KUKA KRL program: MyProgram_181().src

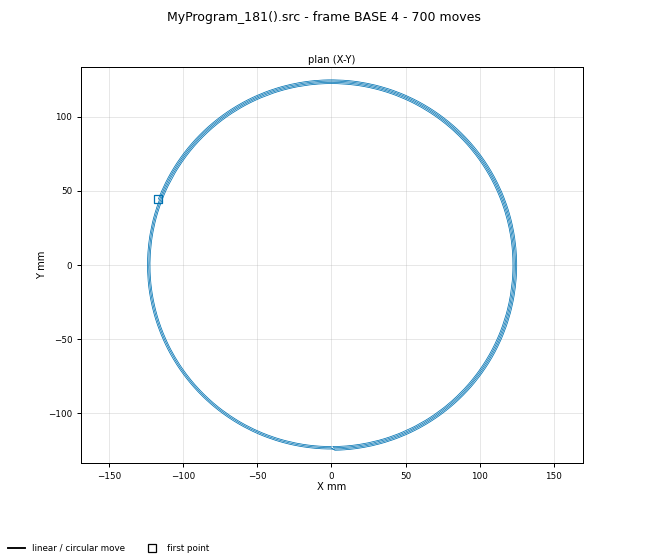
[picture p0: tool path of MyProgram_181().src in frame BASE 4, 700 of 700 moves have a stored position in this frame; points joined in program order, loops and branches not executed]
&ACCESS RVP
&REL 1
&PARAM TEMPLATE = C:\KRC\Roboter\Template\vorgabe
&PARAM EDITMASK = *
DEF MyProgram_181()
; ---- Setting reference (Base) ----
$BASE = BASE_DATA[4]

; --------------------------
; ---- Setting tool (TCP) ----
$TOOL = TOOL_DATA[3]
; --------------------------

$VEL.CP = VEL_APROX_PRINT
Startdeposition()
$VEL.CP = VEL_PRINT
LIN {X -116.6895,Y 44.4583,Z 133,A 155.0312,B 24.9522,C -1.5964,E1 24.8506,E2 291.2943} C_DIS
LIN {X -115.697,Y 46.9762,Z 133,A 153.7111,B 24.9522,C -1.5969,E1 24.852,E2 292.6207} C_DIS
LIN {X -114.3662,Y 50.133,Z 133,A 152.1883,B 24.9518,C -1.6039,E1 24.8537,E2 294.1352} C_DIS
LIN {X -113.0397,Y 53.0574,Z 133,A 150.686,B 24.9516,C -1.6071,E1 24.8554,E2 295.638} C_DIS
LIN {X -111.9021,Y 55.4109,Z 133,A 149.4421,B 24.9516,C -1.6088,E1 24.857,E2 296.8845} C_DIS
LIN {X -110.1873,Y 58.7517,Z 133,A 147.6606,B 24.9513,C -1.6113,E1 24.8593,E2 298.6696} C_DIS
LIN {X -108.2507,Y 62.2485,Z 133,A 145.7452,B 24.9513,C -1.6131,E1 24.8619,E2 300.5907} C_DIS
LIN {X -105.81,Y 66.3134,Z 133,A 143.6874,B 24.9505,C -1.6247,E1 24.8649,E2 302.6316} C_DIS
LIN {X -103.9306,Y 69.2193,Z 133,A 142.0204,B 24.9505,C -1.6257,E1 24.8675,E2 304.3045} C_DIS
LIN {X -101.3647,Y 72.9272,Z 133,A 139.999,B 24.95,C -1.6336,E1 24.8707,E2 306.317} C_DIS
LIN {X -99.2695,Y 75.7526,Z 133,A 138.3169,B 24.95,C -1.635,E1 24.8735,E2 308.0039} C_DIS
LIN {X -96.6511,Y 79.0667,Z 133,A 136.3828,B 24.9496,C -1.6403,E1 24.8769,E2 309.9343} C_DIS
LIN {X -94.1983,Y 81.973,Z 133,A 134.6073,B 24.9494,C -1.6435,E1 24.8801,E2 311.7102} C_DIS
LIN {X -91.6588,Y 84.8038,Z 133,A 132.8618,B 24.9491,C -1.648,E1 24.8834,E2 313.4528} C_DIS
LIN {X -88.8677,Y 87.7247,Z 133,A 130.926,B 24.9491,C -1.6489,E1 24.8872,E2 315.3948} C_DIS
LIN {X -86.0086,Y 90.5292,Z 133,A 129.1473,B 24.9486,C -1.656,E1 24.8907,E2 317.164} C_DIS
LIN {X -83.0096,Y 93.2873,Z 133,A 127.2009,B 24.9486,C -1.6569,E1 24.8948,E2 319.1159} C_DIS
LIN {X -79.9792,Y 95.8975,Z 133,A 125.4366,B 24.9481,C -1.6643,E1 24.8985,E2 320.8696} C_DIS
LIN {X -76.816,Y 98.4502,Z 133,A 123.4845,B 24.9481,C -1.6644,E1 24.9028,E2 322.8286} C_DIS
LIN {X -73.6345,Y 100.8511,Z 133,A 121.7327,B 24.9476,C -1.6718,E1 24.9067,E2 324.5692} C_DIS
LIN {X -70.3577,Y 103.1645,Z 133,A 119.7925,B 24.9476,C -1.671,E1 24.9112,E2 326.5178} C_DIS
LIN {X -66.9879,Y 105.3831,Z 133,A 118.0307,B 24.9472,C -1.6786,E1 24.9153,E2 328.267} C_DIS
LIN {X -63.5914,Y 107.4674,Z 133,A 116.1028,B 24.9472,C -1.6775,E1 24.9199,E2 330.2036} C_DIS
LIN {X -59.4752,Y 109.7995,Z 133,A 113.9327,B 24.947,C -1.6814,E1 24.9252,E2 332.3708} C_DIS
LIN {X -56.3954,Y 111.4096,Z 133,A 112.4464,B 24.9465,C -1.689,E1 24.9289,E2 333.8429} C_DIS
LIN {X -53.3186,Y 112.9163,Z 133,A 110.9027,B 24.9463,C -1.6928,E1 24.9327,E2 335.3817} C_DIS
LIN {X -50.4991,Y 114.2045,Z 133,A 109.4916,B 24.9461,C -1.6955,E1 24.9363,E2 336.7898} C_DIS
LIN {X -47.5925,Y 115.4458,Z 133,A 108.05,B 24.946,C -1.698,E1 24.94,E2 338.2288} C_DIS
LIN {X -44.9062,Y 116.5167,Z 133,A 106.6465,B 24.946,C -1.6963,E1 24.9437,E2 339.6392} C_DIS
LIN {X -41.647,Y 117.7232,Z 133,A 105.0866,B 24.9458,C -1.6999,E1 24.9478,E2 341.1937} C_DIS
LIN {X -38.7891,Y 118.6945,Z 133,A 103.7405,B 24.9456,C -1.7034,E1 24.9513,E2 342.534} C_DIS
LIN {X -36.2059,Y 119.5067,Z 133,A 102.4321,B 24.9457,C -1.7018,E1 24.9548,E2 343.8484} C_DIS
LIN {X -32.9677,Y 120.4422,Z 133,A 100.9122,B 24.9455,C -1.7047,E1 24.9589,E2 345.3639} C_DIS
LIN {X -29.9898,Y 121.2171,Z 133,A 99.5473,B 24.9453,C -1.7083,E1 24.9626,E2 346.7223} C_DIS
LIN {X -27.3572,Y 121.8375,Z 133,A 98.2908,B 24.9453,C -1.7087,E1 24.966,E2 347.9793} C_DIS
LIN {X -24.1727,Y 122.5102,Z 133,A 96.8162,B 24.9451,C -1.7109,E1 24.97,E2 349.4506} C_DIS
LIN {X -21.6943,Y 122.9714,Z 133,A 95.5852,B 24.9453,C -1.7083,E1 24.9734,E2 350.6889} C_DIS
LIN {X -18.3848,Y 123.5119,Z 133,A 94.0677,B 24.9452,C -1.7103,E1 24.9776,E2 352.203} C_DIS
LIN {X -14.9172,Y 123.9758,Z 133,A 92.4267,B 24.9452,C -1.7097,E1 24.9822,E2 353.8466} C_DIS
LIN {X -11.5107,Y 124.3398,Z 133,A 90.8991,B 24.945,C -1.7126,E1 24.9864,E2 355.3683} C_DIS
LIN {X -8.4462,Y 124.5859,Z 133,A 89.5189,B 24.945,C -1.7146,E1 24.9902,E2 356.7442} C_DIS
LIN {X -5.7492,Y 124.7393,Z 133,A 88.2519,B 24.945,C -1.7138,E1 24.9938,E2 358.0135} C_DIS
LIN {X -2.325,Y 124.8487,Z 133,A 86.6375,B 24.945,C -1.7122,E1 24.9983,E2 359.6318} C_DIS
LIN {X 1.3218,Y 124.8654,Z 133,A 84.8045,B 24.9455,C -1.705,E1 25.0034,E2 361.4819} C_DIS
LIN {X 5.505,Y 124.7509,Z 133,A 83.1157,B 24.9448,C -1.7161,E1 25.0081,E2 363.144} C_DIS
LIN {X 8.0461,Y 124.6112,Z 133,A 81.7359,B 24.9455,C -1.7061,E1 25.012,E2 364.5469} C_DIS
LIN {X 11.9921,Y 124.2936,Z 133,A 80.0376,B 24.9451,C -1.7115,E1 25.0167,E2 366.2314} C_DIS
LIN {X 14.8682,Y 123.9817,Z 133,A 78.6941,B 24.9451,C -1.7105,E1 25.0204,E2 367.5763} C_DIS
LIN {X 18.2642,Y 123.5297,Z 133,A 77.174,B 24.9451,C -1.7125,E1 25.0246,E2 369.0903} C_DIS
LIN {X 21.2737,Y 123.0464,Z 133,A 75.8309,B 24.9449,C -1.7147,E1 25.0283,E2 370.4269} C_DIS
LIN {X 23.9077,Y 122.5611,Z 133,A 74.5912,B 24.9449,C -1.7137,E1 25.0317,E2 371.6675} C_DIS
LIN {X 27.0788,Y 121.9008,Z 133,A 73.1177,B 24.9449,C -1.7135,E1 25.0357,E2 373.1395} C_DIS
LIN {X 29.5009,Y 121.3353,Z 133,A 71.8951,B 24.9453,C -1.709,E1 25.039,E2 374.3711} C_DIS
LIN {X 32.8189,Y 120.4825,Z 133,A 70.3477,B 24.9453,C -1.7091,E1 25.0432,E2 375.9158} C_DIS
LIN {X 35.8156,Y 119.6254,Z 133,A 68.9731,B 24.9452,C -1.7108,E1 25.0469,E2 377.2842} C_DIS
LIN {X 38.3543,Y 118.8346,Z 133,A 67.6655,B 24.9455,C -1.7056,E1 25.0504,E2 378.6015} C_DIS
LIN {X 41.6005,Y 117.7396,Z 133,A 66.1321,B 24.9455,C -1.706,E1 25.0544,E2 380.1309} C_DIS
LIN {X 44.4583,Y 116.6895,Z 133,A 64.7708,B 24.9455,C -1.7064,E1 25.058,E2 381.4883} C_DIS
LIN {X 46.9533,Y 115.7063,Z 133,A 63.4699,B 24.9457,C -1.7018,E1 25.0614,E2 382.7974} C_DIS
LIN {X 50.1104,Y 114.376,Z 133,A 61.9635,B 24.9457,C -1.7032,E1 25.0652,E2 384.2968} C_DIS
LIN {X 53.0574,Y 113.0397,Z 133,A 60.4644,B 24.9457,C -1.7007,E1 25.069,E2 385.798} C_DIS
LIN {X 55.4907,Y 111.8627,Z 133,A 59.2079,B 24.9459,C -1.6984,E1 25.0722,E2 387.0566} C_DIS
LIN {X 58.7517,Y 110.1873,Z 133,A 57.4722,B 24.9463,C -1.6935,E1 25.0765,E2 388.7991} C_DIS
LIN {X 62.2484,Y 108.2507,Z 133,A 55.5685,B 24.9466,C -1.6874,E1 25.0811,E2 390.7114} C_DIS
LIN {X 66.3133,Y 105.81,Z 133,A 53.5313,B 24.9464,C -1.6909,E1 25.086,E2 392.7341} C_DIS
LIN {X 69.2398,Y 103.9169,Z 133,A 51.8763,B 24.9468,C -1.6855,E1 25.0898,E2 394.3963} C_DIS
LIN {X 72.9272,Y 101.3646,Z 133,A 49.8782,B 24.9468,C -1.6849,E1 25.0944,E2 396.389} C_DIS
LIN {X 75.7723,Y 99.2545,Z 133,A 48.2058,B 24.9471,C -1.6796,E1 25.0981,E2 398.0676} C_DIS
LIN {X 79.3312,Y 96.4353,Z 133,A 46.1821,B 24.9471,C -1.6786,E1 25.1025,E2 400.0862} C_DIS
LIN {X 81.9916,Y 94.1821,Z 133,A 44.5325,B 24.9476,C -1.673,E1 25.106,E2 401.7426} C_DIS
LIN {X 84.8038,Y 91.6588,Z 133,A 42.8054,B 24.9478,C -1.6697,E1 25.1096,E2 403.4705} C_DIS
LIN {X 87.7247,Y 88.8677,Z 133,A 40.8925,B 24.9482,C -1.6628,E1 25.1135,E2 405.3917} C_DIS
LIN {X 90.5292,Y 86.0086,Z 133,A 39.1388,B 24.9482,C -1.6629,E1 25.1168,E2 407.1376} C_DIS
LIN {X 93.2873,Y 83.0096,Z 133,A 37.2042,B 24.9487,C -1.6554,E1 25.1205,E2 409.0814} C_DIS
LIN {X 95.8975,Y 79.9792,Z 133,A 35.4643,B 24.9487,C -1.6558,E1 25.1236,E2 410.8124} C_DIS
LIN {X 98.4502,Y 76.816,Z 133,A 33.5535,B 24.949,C -1.6489,E1 25.1269,E2 412.7304} C_DIS
LIN {X 100.8511,Y 73.6345,Z 133,A 31.7966,B 24.9491,C -1.648,E1 25.1299,E2 414.4812} C_DIS
LIN {X 103.1645,Y 70.3577,Z 133,A 29.8671,B 24.9497,C -1.6387,E1 25.1329,E2 416.423} C_DIS
LIN {X 105.3831,Y 66.9879,Z 133,A 28.1306,B 24.9497,C -1.6396,E1 25.1356,E2 418.1487} C_DIS
LIN {X 107.4674,Y 63.5914,Z 133,A 26.2144,B 24.9502,C -1.6303,E1 25.1383,E2 420.0772} C_DIS
LIN {X 109.8114,Y 59.4535,Z 133,A 24.0555,B 24.9505,C -1.6254,E1 25.1413,E2 422.2363} C_DIS
LIN {X 112.1236,Y 54.9624,Z 133,A 21.8943,B 24.9505,C -1.6268,E1 25.144,E2 424.3827} C_DIS
LIN {X 113.6675,Y 51.6979,Z 133,A 20.282,B 24.9505,C -1.6243,E1 25.1459,E2 425.9923} C_DIS
LIN {X 114.7933,Y 49.1453,Z 133,A 18.9532,B 24.9509,C -1.618,E1 25.1474,E2 427.3284} C_DIS
LIN {X 116.0423,Y 46.1217,Z 133,A 17.4924,B 24.9511,C -1.6156,E1 25.1489,E2 428.7869} C_DIS
LIN {X 117.2068,Y 43.0763,Z 133,A 16.052,B 24.9511,C -1.614,E1 25.1503,E2 430.2232} C_DIS
LIN {X 118.0998,Y 40.5602,Z 133,A 14.7553,B 24.9516,C -1.6066,E1 25.1515,E2 431.5298} C_DIS
LIN {X 119.0422,Y 37.7053,Z 133,A 13.4155,B 24.9518,C -1.6044,E1 25.1526,E2 432.8673} C_DIS
LIN {X 120.0332,Y 34.4239,Z 133,A 11.8937,B 24.9519,C -1.6022,E1 25.1538,E2 434.3858} C_DIS
LIN {X 121.0581,Y 30.6172,Z 133,A 10.0158,B 24.9525,C -1.593,E1 25.1552,E2 436.2744} C_DIS
LIN {X 121.8429,Y 27.3332,Z 133,A 8.5584,B 24.9525,C -1.5928,E1 25.1561,E2 437.7237} C_DIS
LIN {X 122.5102,Y 24.1727,Z 133,A 7.1037,B 24.9527,C -1.5895,E1 25.1569,E2 439.1778} C_DIS
LIN {X 122.9405,Y 21.8675,Z 133,A 5.9294,B 24.9532,C -1.5811,E1 25.1575,E2 440.3651} C_DIS
LIN {X 123.5119,Y 18.3848,Z 133,A 4.398,B 24.9532,C -1.5803,E1 25.1582,E2 441.8892} C_DIS
LIN {X 124.0763,Y 14.0747,Z 133,A 2.4493,B 24.9534,C -1.5763,E1 25.1589,E2 443.836} C_DIS
LIN {X 124.3421,Y 11.4861,Z 133,A 1.2276,B 24.9538,C -1.571,E1 25.1592,E2 445.063} C_DIS
LIN {X 124.5859,Y 8.4462,Z 133,A -0.1347,B 24.9539,C -1.5683,E1 25.1595,E2 446.4235} C_DIS
LIN {X 124.7483,Y 5.5668,Z 133,A -1.6675,B 24.9548,C -1.5532,E1 25.1597,E2 447.9827} C_DIS
LIN {X 124.8637,Y 1.4441,Z 133,A -3.3231,B 24.9545,C -1.5592,E1 25.1597,E2 449.6145} C_DIS
LIN {X 124.8646,Y -1.3828,Z 133,A -4.8305,B 24.9553,C -1.5441,E1 25.1597,E2 451.1484} C_DIS
LIN {X 124.7508,Y -5.505,Z 133,A -6.489,B 24.955,C -1.5499,E1 25.1596,E2 452.7834} C_DIS
LIN {X 124.5347,Y -9.1442,Z 133,A -8.2497,B 24.9556,C -1.5399,E1 25.1593,E2 454.5571} C_DIS
LIN {X 124.2394,Y -12.5574,Z 133,A -9.7621,B 24.9556,C -1.5378,E1 25.1589,E2 456.0656} C_DIS
LIN {X 123.9788,Y -14.8927,Z 133,A -10.8875,B 24.956,C -1.5318,E1 25.1585,E2 457.1984} C_DIS
LIN {X 123.5851,Y -17.8742,Z 133,A -12.2192,B 24.9562,C -1.5298,E1 25.158,E2 458.5271} C_DIS
LIN {X 123.1574,Y -20.6093,Z 133,A -13.5143,B 24.9565,C -1.5243,E1 25.1574,E2 459.8274} C_DIS
LIN {X 122.5658,Y -23.8834,Z 133,A -14.9527,B 24.9565,C -1.5239,E1 25.1567,E2 461.2584} C_DIS
LIN {X 121.9008,Y -27.0788,Z 133,A -16.4252,B 24.9567,C -1.5203,E1 25.1558,E2 462.731} C_DIS
LIN {X 121.3295,Y -29.5249,Z 133,A -17.6476,B 24.9571,C -1.513,E1 25.155,E2 463.9634} C_DIS
LIN {X 120.5319,Y -32.6336,Z 133,A -19.0811,B 24.9573,C -1.5102,E1 25.154,E2 465.3953} C_DIS
LIN {X 119.6254,Y -35.8156,Z 133,A -20.5468,B 24.9573,C -1.508,E1 25.1529,E2 466.8578} C_DIS
LIN {X 118.8421,Y -38.3307,Z 133,A -21.838,B 24.9579,C -1.4999,E1 25.1518,E2 468.1606} C_DIS
LIN {X 117.7477,Y -41.5771,Z 133,A -23.3597,B 24.9579,C -1.4975,E1 25.1504,E2 469.6795} C_DIS
LIN {X 116.6895,Y -44.4583,Z 133,A -24.7286,B 24.9581,C -1.4951,E1 25.1491,E2 471.0464} C_DIS
LIN {X 115.697,Y -46.9762,Z 133,A -25.9971,B 24.9584,C -1.4898,E1 25.1477,E2 472.3203} C_DIS
LIN {X 114.3662,Y -50.133,Z 133,A -27.5341,B 24.9586,C -1.4867,E1 25.146,E2 473.8562} C_DIS
LIN {X 113.0397,Y -53.0574,Z 133,A -29.0168,B 24.9589,C -1.4817,E1 25.1443,E2 475.3427} C_DIS
LIN {X 111.924,Y -55.3666,Z 133,A -30.2101,B 24.9591,C -1.4773,E1 25.1428,E2 476.5399} C_DIS
LIN {X 110.1873,Y -58.7517,Z 133,A -32.0034,B 24.9595,C -1.4696,E1 25.1405,E2 478.3421} C_DIS
LIN {X 108.2507,Y -62.2485,Z 133,A -33.8947,B 24.96,C -1.4612,E1 25.1379,E2 480.2432} C_DIS
LIN {X 105.81,Y -66.3134,Z 133,A -35.9274,B 24.96,C -1.4621,E1 25.1349,E2 482.2634} C_DIS
LIN {X 103.9306,Y -69.2193,Z 133,A -37.5741,B 24.9604,C -1.4546,E1 25.1324,E2 483.9196} C_DIS
LIN {X 101.3647,Y -72.9272,Z 133,A -39.5716,B 24.9604,C -1.4524,E1 25.1292,E2 485.9125} C_DIS
LIN {X 99.2695,Y -75.7526,Z 133,A -41.234,B 24.9609,C -1.4455,E1 25.1264,E2 487.5834} C_DIS
LIN {X 96.4353,Y -79.3313,Z 133,A -43.2607,B 24.9609,C -1.4433,E1 25.1229,E2 489.6059} C_DIS
LIN {X 94.1983,Y -81.973,Z 133,A -44.9018,B 24.9613,C -1.4364,E1 25.1199,E2 491.2556} C_DIS
LIN {X 91.6588,Y -84.8038,Z 133,A -46.6283,B 24.9615,C -1.4328,E1 25.1166,E2 492.9829} C_DIS
LIN {X 88.8677,Y -87.7247,Z 133,A -48.5435,B 24.962,C -1.4251,E1 25.1129,E2 494.9082} C_DIS
LIN {X 86.0086,Y -90.5292,Z 133,A -50.304,B 24.962,C -1.4245,E1 25.1093,E2 496.6629} C_DIS
LIN {X 83.0096,Y -93.2873,Z 133,A -52.2308,B 24.9624,C -1.4171,E1 25.1053,E2 498.5992} C_DIS
LIN {X 79.9792,Y -95.8975,Z 133,A -53.9782,B 24.9624,C -1.4174,E1 25.1016,E2 500.3393} C_DIS
LIN {X 76.816,Y -98.4502,Z 133,A -55.9119,B 24.9628,C -1.4097,E1 25.0974,E2 502.2837} C_DIS
LIN {X 73.6345,Y -100.8511,Z 133,A -57.6481,B 24.9628,C -1.4105,E1 25.0935,E2 504.012} C_DIS
LIN {X 70.3577,Y -103.1645,Z 133,A -59.5713,B 24.9632,C -1.4025,E1 25.0891,E2 505.9473} C_DIS
LIN {X 66.9879,Y -105.3831,Z 133,A -61.3186,B 24.9631,C -1.4041,E1 25.085,E2 507.6852} C_DIS
LIN {X 63.5914,Y -107.4674,Z 133,A -63.231,B 24.9635,C -1.3964,E1 25.0804,E2 509.6099} C_DIS
LIN {X 59.4752,Y -109.7995,Z 133,A -65.3847,B 24.9636,C -1.3934,E1 25.0751,E2 511.7645} C_DIS
LIN {X 56.3954,Y -111.4096,Z 133,A -66.8606,B 24.9635,C -1.3966,E1 25.0715,E2 513.2286} C_DIS
LIN {X 53.3186,Y -112.9163,Z 133,A -68.3983,B 24.9635,C -1.3957,E1 25.0676,E2 514.7644} C_DIS
LIN {X 50.2713,Y -114.3064,Z 133,A -69.9153,B 24.9635,C -1.3943,E1 25.0637,E2 516.281} C_DIS
LIN {X 47.4675,Y -115.498,Z 133,A -71.2814,B 24.9636,C -1.3938,E1 25.0602,E2 517.6449} C_DIS
LIN {X 44.9062,Y -116.5167,Z 133,A -72.6234,B 24.9639,C -1.3882,E1 25.0567,E2 518.9972} C_DIS
LIN {X 41.647,Y -117.7232,Z 133,A -74.1722,B 24.9639,C -1.3883,E1 25.0527,E2 520.5426} C_DIS
LIN {X 38.7891,Y -118.6945,Z 133,A -75.5018,B 24.9639,C -1.3894,E1 25.0492,E2 521.8673} C_DIS
LIN {X 36.2059,Y -119.5067,Z 133,A -76.8155,B 24.9641,C -1.3844,E1 25.0456,E2 523.1904} C_DIS
LIN {X 32.9677,Y -120.4422,Z 133,A -78.3284,B 24.9641,C -1.3843,E1 25.0416,E2 524.701} C_DIS
LIN {X 29.9898,Y -121.2171,Z 133,A -79.6875,B 24.9641,C -1.3854,E1 25.0379,E2 526.0553} C_DIS
LIN {X 27.3572,Y -121.8375,Z 133,A -80.9389,B 24.9641,C -1.3837,E1 25.0345,E2 527.309} C_DIS
LIN {X 24.1727,Y -122.5102,Z 133,A -82.4081,B 24.9641,C -1.3836,E1 25.0305,E2 528.7767} C_DIS
LIN {X 21.6943,Y -122.9714,Z 133,A -83.6348,B 24.9644,C -1.3792,E1 25.0271,E2 530.0124} C_DIS
LIN {X 18.6063,Y -123.4775,Z 133,A -85.0343,B 24.9644,C -1.3799,E1 25.0232,E2 531.4089} C_DIS
LIN {X 16.0341,Y -123.8366,Z 133,A -86.203,B 24.9644,C -1.3803,E1 25.02,E2 532.5757} C_DIS
LIN {X 12.7087,Y -124.2243,Z 133,A -87.7444,B 24.9644,C -1.3791,E1 25.0157,E2 534.119} C_DIS
LIN {X 8.6784,Y -124.5689,Z 133,A -89.5972,B 24.9644,C -1.3783,E1 25.0105,E2 535.9725} C_DIS
LIN {X 5.7492,Y -124.7393,Z 133,A -90.9508,B 24.9644,C -1.3774,E1 25.0068,E2 537.3279} C_DIS
LIN {X 2.325,Y -124.8487,Z 133,A -92.5631,B 24.9646,C -1.375,E1 25.0023,E2 538.9456} C_DIS
LIN {X 2.325,Y -124.8487,Z 133,A -92.5631,B 24.9646,C -1.375,E1 25.0023,E2 538.9456} C_DIS
Enddeposition()
LIN {X 0.8859,Y -124.0293,Z 133,A -93.2093,B 24.9638,C -1.3903,E1 25.0006,E2 539.5556} C_DIS
Startdeposition()
$VEL.CP = VEL_PRINT
LIN {X 3.5558,Y -123.9822,Z 133,A -91.4139,B 24.9623,C -1.4178,E1 25.0058,E2 537.6952} C_DIS
LIN {X 6.3715,Y -123.8705,Z 133,A -90.0135,B 24.9621,C -1.4231,E1 25.0097,E2 536.2827} C_DIS
LIN {X 9.98,Y -123.6317,Z 133,A -88.2827,B 24.9619,C -1.4268,E1 25.0145,E2 534.5439} C_DIS
LIN {X 13.8144,Y -123.2627,Z 133,A -86.4414,B 24.9616,C -1.4309,E1 25.0197,E2 532.6943} C_DIS
LIN {X 17.6544,Y -122.7711,Z 133,A -84.7834,B 24.9619,C -1.4257,E1 25.0242,E2 531.0499} C_DIS
LIN {X 21.7768,Y -122.1067,Z 133,A -82.9831,B 24.9622,C -1.4208,E1 25.0291,E2 529.2629} C_DIS
LIN {X 24.7936,Y -121.5298,Z 133,A -81.504,B 24.962,C -1.425,E1 25.0332,E2 527.7757} C_DIS
LIN {X 27.7732,Y -120.8845,Z 133,A -80.0201,B 24.9617,C -1.4301,E1 25.0373,E2 526.2818} C_DIS
LIN {X 31.1769,Y -120.0529,Z 133,A -78.1591,B 24.961,C -1.4438,E1 25.0424,E2 524.3912} C_DIS
LIN {X 34.9694,Y -119.0013,Z 133,A -76.6182,B 24.9616,C -1.4321,E1 25.0464,E2 522.8806} C_DIS
LIN {X 38.0799,Y -118.0438,Z 133,A -74.9694,B 24.9611,C -1.4411,E1 25.0509,E2 521.2135} C_DIS
LIN {X 41.8289,Y -116.7678,Z 133,A -73.2082,B 24.9611,C -1.4401,E1 25.0555,E2 519.4582} C_DIS
LIN {X 45.1339,Y -115.5304,Z 133,A -71.6275,B 24.9611,C -1.4399,E1 25.0596,E2 517.8814} C_DIS
LIN {X 48.4667,Y -114.1737,Z 133,A -69.8642,B 24.9608,C -1.4474,E1 25.0642,E2 516.1045} C_DIS
LIN {X 52.5572,Y -112.3489,Z 133,A -67.8625,B 24.9608,C -1.4473,E1 25.0693,E2 514.1081} C_DIS
LIN {X 57.0107,Y -110.1577,Z 133,A -65.6711,B 24.9608,C -1.446,E1 25.0747,E2 511.9256} C_DIS
LIN {X 61.6993,Y -107.6005,Z 133,A -62.7982,B 24.9595,C -1.471,E1 25.0818,E2 509.0022} C_DIS
LIN {X 64.8534,Y -105.729,Z 133,A -61.5813,B 24.9606,C -1.4501,E1 25.0846,E2 507.8386} C_DIS
LIN {X 67.8771,Y -103.8154,Z 133,A -59.3711,B 24.9589,C -1.4816,E1 25.09,E2 505.5612} C_DIS
LIN {X 71.2509,Y -101.528,Z 133,A -58.093,B 24.9604,C -1.4547,E1 25.0927,E2 504.3509} C_DIS
LIN {X 74.1934,Y -99.3988,Z 133,A -56.216,B 24.9596,C -1.4684,E1 25.097,E2 502.4483} C_DIS
LIN {X 77.4252,Y -96.9017,Z 133,A -54.1352,B 24.9588,C -1.4825,E1 25.1016,E2 500.342} C_DIS
LIN {X 79.9254,Y -94.8499,Z 133,A -52.8711,B 24.9593,C -1.4742,E1 25.1043,E2 499.1023} C_DIS
LIN {X 83.1574,Y -92.0304,Z 133,A -50.8978,B 24.9591,C -1.4784,E1 25.1084,E2 497.1269} C_DIS
LIN {X 86.6144,Y -88.7849,Z 133,A -48.4884,B 24.9581,C -1.4949,E1 25.1133,E2 494.6885} C_DIS
LIN {X 88.9161,Y -86.4791,Z 133,A -46.7364,B 24.9572,C -1.5115,E1 25.1168,E2 492.905} C_DIS
LIN {X 92.0187,Y -83.1704,Z 133,A -45.3655,B 24.959,C -1.4797,E1 25.1192,E2 491.6153} C_DIS
LIN {X 94.2078,Y -80.6831,Z 133,A -43.5512,B 24.9579,C -1.4982,E1 25.1226,E2 489.7654} C_DIS
LIN {X 99.1932,Y -74.4686,Z 133,A -40.0644,B 24.9579,C -1.4982,E1 25.1286,E2 486.2949} C_DIS
LIN {X 101.1843,Y -71.7386,Z 133,A -38.3986,B 24.9574,C -1.508,E1 25.1313,E2 484.6141} C_DIS
LIN {X 103.7575,Y -67.9649,Z 133,A -36.2868,B 24.9571,C -1.5141,E1 25.1346,E2 482.4984} C_DIS
LIN {X 106.0577,Y -64.3145,Z 133,A -34.3457,B 24.9569,C -1.5172,E1 25.1374,E2 480.5598} C_DIS
LIN {X 108.866,Y -59.4378,Z 133,A -31.7507,B 24.9564,C -1.5247,E1 25.141,E2 477.9607} C_DIS
LIN {X 110.4663,Y -56.4043,Z 133,A -30.2235,B 24.9564,C -1.5266,E1 25.143,E2 476.4372} C_DIS
LIN {X 112.1094,Y -53.0661,Z 133,A -28.5971,B 24.9564,C -1.527,E1 25.1449,E2 474.8184} C_DIS
LIN {X 113.5497,Y -49.9129,Z 133,A -26.7086,B 24.9552,C -1.5468,E1 25.1471,E2 472.8936} C_DIS
LIN {X 115.0838,Y -46.2601,Z 133,A -25.1254,B 24.9556,C -1.5398,E1 25.1488,E2 471.3356} C_DIS
LIN {X 116.5902,Y -42.3211,Z 133,A -22.5573,B 24.9533,C -1.5781,E1 25.1513,E2 468.6914} C_DIS
LIN {X 118.1658,Y -37.6984,Z 133,A -21.1923,B 24.9556,C -1.5391,E1 25.1524,E2 467.4263} C_DIS
LIN {X 118.947,Y -35.1547,Z 133,A -19.7275,B 24.9547,C -1.5552,E1 25.1536,E2 465.9319} C_DIS
LIN {X 119.9648,Y -31.5112,Z 133,A -17.7372,B 24.9536,C -1.5734,E1 25.1551,E2 463.9101} C_DIS
LIN {X 120.9703,Y -27.3964,Z 133,A -15.9606,B 24.9538,C -1.5704,E1 25.1562,E2 462.1509} C_DIS
LIN {X 121.9265,Y -22.7744,Z 133,A -13.9465,B 24.9538,C -1.5689,E1 25.1573,E2 460.1521} C_DIS
LIN {X 122.3948,Y -20.0956,Z 133,A -12.7048,B 24.9537,C -1.5723,E1 25.1578,E2 458.9097} C_DIS
LIN {X 122.9518,Y -16.3453,Z 133,A -10.6973,B 24.9526,C -1.5913,E1 25.1586,E2 456.8692} C_DIS
LIN {X 123.3707,Y -12.8176,Z 133,A -9.1701,B 24.9526,C -1.5907,E1 25.1591,E2 455.3523} C_DIS
LIN {X 123.6944,Y -9.1605,Z 133,A -7.5598,B 24.9526,C -1.5919,E1 25.1594,E2 453.7488} C_DIS
LIN {X 123.9124,Y -5.5254,Z 133,A -5.79,B 24.9519,C -1.6019,E1 25.1597,E2 451.9659} C_DIS
LIN {X 124.0303,Y -1.1139,Z 133,A -3.8363,B 24.9518,C -1.6042,E1 25.1597,E2 450.0185} C_DIS
LIN {X 124.0095,Y 2.4534,Z 133,A -2.3173,B 24.9518,C -1.603,E1 25.1597,E2 448.5114} C_DIS
LIN {X 123.8912,Y 5.9529,Z 133,A -0.6589,B 24.9514,C -1.6104,E1 25.1595,E2 446.8453} C_DIS
LIN {X 123.6626,Y 9.5941,Z 133,A 1.0564,B 24.951,C -1.6174,E1 25.1592,E2 445.1237} C_DIS
LIN {X 123.3513,Y 12.9962,Z 133,A 2.4302,B 24.9513,C -1.612,E1 25.1588,E2 443.7707} C_DIS
LIN {X 123.0151,Y 15.8622,Z 133,A 3.8699,B 24.9507,C -1.6218,E1 25.1583,E2 442.3164} C_DIS
LIN {X 122.5217,Y 19.3088,Z 133,A 5.486,B 24.9504,C -1.6274,E1 25.1577,E2 440.6967} C_DIS
LIN {X 121.7898,Y 23.4864,Z 133,A 7.9703,B 24.9483,C -1.6608,E1 25.1564,E2 438.1482} C_DIS
LIN {X 120.9086,Y 27.6672,Z 133,A 9.3663,B 24.9498,C -1.6372,E1 25.1556,E2 436.8161} C_DIS
LIN {X 120.1497,Y 30.7951,Z 133,A 10.8555,B 24.9495,C -1.642,E1 25.1545,E2 435.3241} C_DIS
LIN {X 118.7254,Y 35.899,Z 133,A 13.3527,B 24.9489,C -1.652,E1 25.1526,E2 432.8175} C_DIS
LIN {X 117.6528,Y 39.2679,Z 133,A 14.9177,B 24.9488,C -1.6536,E1 25.1513,E2 431.2578} C_DIS
LIN {X 116.6813,Y 42.0688,Z 133,A 16.3181,B 24.9484,C -1.6593,E1 25.1499,E2 429.8518} C_DIS
LIN {X 115.5152,Y 45.1731,Z 133,A 17.8908,B 24.948,C -1.6659,E1 25.1484,E2 428.2722} C_DIS
LIN {X 114.0858,Y 48.6732,Z 133,A 19.6391,B 24.9477,C -1.6711,E1 25.1465,E2 426.5211} C_DIS
LIN {X 111.4188,Y 54.4996,Z 133,A 22.6482,B 24.947,C -1.6822,E1 25.1429,E2 423.5022} C_DIS
LIN {X 109.803,Y 57.6851,Z 133,A 24.1283,B 24.9472,C -1.6782,E1 25.141,E2 422.0395} C_DIS
LIN {X 107.8139,Y 61.3259,Z 133,A 26.1659,B 24.9465,C -1.6896,E1 25.1382,E2 419.9855} C_DIS
LIN {X 105.4931,Y 65.2374,Z 133,A 28.175,B 24.9465,C -1.6906,E1 25.1353,E2 417.9843} C_DIS
LIN {X 103.3371,Y 68.6012,Z 133,A 30.0123,B 24.9462,C -1.695,E1 25.1325,E2 416.1457} C_DIS
LIN {X 101.1257,Y 71.8217,Z 133,A 31.5892,B 24.9466,C -1.6881,E1 25.13,E2 414.5928} C_DIS
LIN {X 99.16,Y 74.5126,Z 133,A 33.4363,B 24.9454,C -1.7076,E1 25.1269,E2 412.7087} C_DIS
LIN {X 93.8986,Y 81.0415,Z 133,A 36.8985,B 24.9461,C -1.6961,E1 25.1209,E2 409.2896} C_DIS
LIN {X 91.4285,Y 83.8176,Z 133,A 38.9118,B 24.9449,C -1.715,E1 25.117,E2 407.2408} C_DIS
LIN {X 88.6849,Y 86.7162,Z 133,A 40.7508,B 24.9446,C -1.7188,E1 25.1135,E2 405.4005} C_DIS
LIN {X 82.3107,Y 92.788,Z 133,A 44.6184,B 24.9447,C -1.7173,E1 25.1057,E2 401.5525} C_DIS
LIN {X 79.577,Y 95.1425,Z 133,A 46.4597,B 24.944,C -1.7293,E1 25.1017,E2 399.69} C_DIS
LIN {X 76.428,Y 97.6907,Z 133,A 48.2789,B 24.9439,C -1.7302,E1 25.0977,E2 397.8754} C_DIS
LIN {X 73.4502,Y 99.9481,Z 133,A 50.0816,B 24.9434,C -1.7371,E1 25.0937,E2 396.0628} C_DIS
LIN {X 69.884,Y 102.4746,Z 133,A 52.0902,B 24.9433,C -1.74,E1 25.0891,E2 394.0543} C_DIS
LIN {X 66.4489,Y 104.734,Z 133,A 53.9827,B 24.9431,C -1.7428,E1 25.0846,E2 392.1615} C_DIS
LIN {X 62.6592,Y 107.044,Z 133,A 55.885,B 24.9434,C -1.7386,E1 25.0801,E2 390.275} C_DIS
LIN {X 59.275,Y 108.9551,Z 133,A 57.8558,B 24.9426,C -1.7498,E1 25.0752,E2 388.2835} C_DIS
LIN {X 55.3777,Y 110.9852,Z 133,A 59.9211,B 24.9423,C -1.7542,E1 25.0701,E2 386.2134} C_DIS
LIN {X 51.3378,Y 112.9119,Z 133,A 61.7646,B 24.9429,C -1.7456,E1 25.0655,E2 384.3947} C_DIS
LIN {X 48.3344,Y 114.229,Z 133,A 63.5089,B 24.942,C -1.7586,E1 25.0609,E2 382.6241} C_DIS
LIN {X 43.9336,Y 115.9923,Z 133,A 65.5764,B 24.9423,C -1.7548,E1 25.0556,E2 380.5701} C_DIS
LIN {X 40.1406,Y 117.3595,Z 133,A 67.3385,B 24.9425,C -1.7516,E1 25.051,E2 378.8192} C_DIS
LIN {X 34.3616,Y 119.1794,Z 133,A 70.0646,B 24.9425,C -1.7502,E1 25.0437,E2 376.1013} C_DIS
LIN {X 31.5406,Y 119.957,Z 133,A 71.7954,B 24.9413,C -1.7694,E1 25.0389,E2 374.3276} C_DIS
LIN {X 26.7398,Y 121.1179,Z 133,A 73.8442,B 24.942,C -1.7594,E1 25.0334,E2 372.3054} C_DIS
LIN {X 22.9306,Y 121.8965,Z 133,A 75.5899,B 24.942,C -1.7577,E1 25.0287,E2 370.5657} C_DIS
LIN {X 18.4276,Y 122.6584,Z 133,A 77.6255,B 24.9423,C -1.7549,E1 25.0231,E2 368.5388} C_DIS
LIN {X 15.0746,Y 123.1143,Z 133,A 79.2629,B 24.942,C -1.7588,E1 25.0185,E2 366.8934} C_DIS
LIN {X 11.716,Y 123.4794,Z 133,A 80.8193,B 24.942,C -1.7588,E1 25.0142,E2 365.3381} C_DIS
LIN {X 8.3403,Y 123.7544,Z 133,A 82.526,B 24.9416,C -1.7657,E1 25.0094,E2 363.6159} C_DIS
LIN {X 5.0114,Y 123.9324,Z 133,A 83.9197,B 24.942,C -1.7586,E1 25.0056,E2 362.2394} C_DIS
LIN {X 1.0086,Y 124.0303,Z 133,A 85.7913,B 24.942,C -1.7594,E1 25.0003,E2 360.3661} C_DIS
LIN {X -2.6617,Y 124.006,Z 133,A 87.5064,B 24.942,C -1.7599,E1 24.9955,E2 358.6498} C_DIS
LIN {X -6.6373,Y 123.8573,Z 133,A 89.4432,B 24.9417,C -1.764,E1 24.9901,E2 356.7029} C_DIS
LIN {X -10.7031,Y 123.571,Z 133,A 91.253,B 24.942,C -1.7597,E1 24.9851,E2 354.9025} C_DIS
LIN {X -14.7477,Y 123.1533,Z 133,A 93.0653,B 24.9422,C -1.7555,E1 24.9801,E2 353.0989} C_DIS
LIN {X -19.7935,Y 122.4452,Z 133,A 95.3399,B 24.9426,C -1.7502,E1 24.9738,E2 350.8351} C_DIS
LIN {X -28.1635,Y 120.7956,Z 133,A 99.3624,B 24.9426,C -1.7506,E1 24.9628,E2 346.807} C_DIS
LIN {X -32.338,Y 119.7446,Z 133,A 101.5073,B 24.9422,C -1.7559,E1 24.957,E2 344.6464} C_DIS
LIN {X -36.19,Y 118.6364,Z 133,A 103.3087,B 24.9425,C -1.7515,E1 24.9522,E2 342.8524} C_DIS
LIN {X -40.4709,Y 117.2451,Z 133,A 105.9696,B 24.9409,C -1.776,E1 24.945,E2 340.1281} C_DIS
LIN {X -45.0709,Y 115.5549,Z 133,A 107.5069,B 24.9433,C -1.7392,E1 24.9412,E2 338.6751} C_DIS
LIN {X -47.4506,Y 114.5982,Z 133,A 108.8036,B 24.9431,C -1.7426,E1 24.9378,E2 337.3673} C_DIS
LIN {X -50.8002,Y 113.1529,Z 133,A 110.7175,B 24.9426,C -1.7507,E1 24.9329,E2 335.4297} C_DIS
LIN {X -55.1327,Y 111.1062,Z 133,A 112.6255,B 24.9437,C -1.733,E1 24.9282,E2 333.5587} C_DIS
LIN {X -58.5811,Y 109.3294,Z 133,A 114.5844,B 24.9434,C -1.7376,E1 24.9233,E2 331.5834} C_DIS
LIN {X -62.257,Y 107.2783,Z 133,A 116.4586,B 24.9438,C -1.7309,E1 24.9188,E2 329.7197} C_DIS
LIN {X -65.6502,Y 105.2367,Z 133,A 118.4096,B 24.9438,C -1.733,E1 24.9141,E2 327.7576} C_DIS
LIN {X -69.5314,Y 102.7131,Z 133,A 120.4881,B 24.9442,C -1.7261,E1 24.9093,E2 325.6888} C_DIS
LIN {X -72.9755,Y 100.2956,Z 133,A 122.4562,B 24.9444,C -1.7232,E1 24.9048,E2 323.7208} C_DIS
LIN {X -76.5034,Y 97.6315,Z 133,A 124.5347,B 24.9445,C -1.7204,E1 24.9002,E2 321.6412} C_DIS
LIN {X -79.6512,Y 95.0802,Z 133,A 126.3504,B 24.945,C -1.7137,E1 24.8963,E2 319.8347} C_DIS
LIN {X -82.9389,Y 92.2273,Z 133,A 128.4243,B 24.945,C -1.7119,E1 24.892,E2 317.7569} C_DIS
LIN {X -86.074,Y 89.3079,Z 133,A 130.3916,B 24.9454,C -1.7066,E1 24.888,E2 315.7939} C_DIS
LIN {X -89.092,Y 86.2974,Z 133,A 132.3606,B 24.9457,C -1.7018,E1 24.8841,E2 313.8282} C_DIS
LIN {X -92.0675,Y 83.1168,Z 133,A 134.4273,B 24.9459,C -1.6991,E1 24.8802,E2 311.7587} C_DIS
LIN {X -94.7666,Y 80.0249,Z 133,A 136.3261,B 24.9462,C -1.6943,E1 24.8768,E2 309.8627} C_DIS
LIN {X -97.4905,Y 76.6829,Z 133,A 138.3002,B 24.9466,C -1.6881,E1 24.8733,E2 307.894} C_DIS
LIN {X -99.9533,Y 73.4431,Z 133,A 140.1542,B 24.947,C -1.6818,E1 24.8703,E2 306.0461} C_DIS
LIN {X -102.5748,Y 69.7362,Z 133,A 142.226,B 24.9474,C -1.6748,E1 24.867,E2 303.9809} C_DIS
LIN {X -104.5452,Y 66.7449,Z 133,A 143.885,B 24.9477,C -1.6703,E1 24.8644,E2 302.3242} C_DIS
LIN {X -106.7152,Y 63.2189,Z 133,A 145.8353,B 24.948,C -1.6664,E1 24.8616,E2 300.3732} C_DIS
LIN {X -108.4898,Y 60.1209,Z 133,A 147.467,B 24.9483,C -1.6608,E1 24.8594,E2 298.7463} C_DIS
LIN {X -110.1607,Y 57.005,Z 133,A 149.4146,B 24.9477,C -1.6699,E1 24.8568,E2 296.7667} C_DIS
LIN {X -112.0866,Y 53.1137,Z 133,A 151.0986,B 24.949,C -1.6495,E1 24.8548,E2 295.1222} C_DIS
LIN {X -113.3254,Y 50.4146,Z 133,A 152.5167,B 24.9491,C -1.6473,E1 24.8532,E2 293.7014} C_DIS
LIN {X -115.0123,Y 46.4369,Z 133,A 154.5962,B 24.9493,C -1.6449,E1 24.851,E2 291.6162} C_DIS
LIN {X -116.4149,Y 42.8047,Z 133,A 156.4474,B 24.9495,C -1.6415,E1 24.8492,E2 289.7625} C_DIS
LIN {X -117.6385,Y 39.3108,Z 133,A 158.11,B 24.95,C -1.634,E1 24.8477,E2 288.1083} C_DIS
LIN {X -119.0141,Y 34.9257,Z 133,A 160.1791,B 24.9505,C -1.6249,E1 24.846,E2 286.0492} C_DIS
LIN {X -119.9113,Y 31.7122,Z 133,A 161.706,B 24.9509,C -1.6193,E1 24.8449,E2 284.5267} C_DIS
LIN {X -120.7064,Y 28.5408,Z 133,A 163.4001,B 24.9507,C -1.6225,E1 24.8437,E2 282.815} C_DIS
LIN {X -122.1749,Y 21.3941,Z 133,A 166.5462,B 24.9519,C -1.6016,E1 24.8421,E2 279.7002} C_DIS
LIN {X -122.6148,Y 18.709,Z 133,A 168.178,B 24.9512,C -1.6141,E1 24.8413,E2 278.0288} C_DIS
LIN {X -123.1938,Y 14.4073,Z 133,A 169.8826,B 24.9524,C -1.5942,E1 24.8408,E2 276.3614} C_DIS
LIN {X -123.5038,Y 11.4615,Z 133,A 171.3058,B 24.9525,C -1.5921,E1 24.8404,E2 274.9347} C_DIS
LIN {X -123.7427,Y 8.5024,Z 133,A 172.8011,B 24.9525,C -1.5931,E1 24.8401,E2 273.4279} C_DIS
LIN {X -124.0018,Y 2.8572,Z 133,A 175.4499,B 24.9529,C -1.5863,E1 24.8398,E2 270.7796} C_DIS
LIN {X -123.9758,Y -3.7863,Z 133,A 177.9877,B 24.9548,C -1.5527,E1 24.8398,E2 268.3066} C_DIS
LIN {X -123.5574,Y -10.8648,Z 133,A -178.3715,B 24.9545,C -1.5581,E1 24.8405,E2 264.631} C_DIS
LIN {X -123.1186,Y -15.0385,Z 133,A -176.045,B 24.9539,C -1.5691,E1 24.8412,E2 262.2642} C_DIS
LIN {X -122.6875,Y -18.2394,Z 133,A -174.2558,B 24.9534,C -1.5776,E1 24.842,E2 260.4441} C_DIS
LIN {X -121.9566,Y -22.617,Z 133,A -172.6072,B 24.9548,C -1.5531,E1 24.8428,E2 258.8442} C_DIS
LIN {X -121.1902,Y -26.4046,Z 133,A -171.0469,B 24.9557,C -1.5374,E1 24.8437,E2 257.312} C_DIS
LIN {X -120.5423,Y -29.2196,Z 133,A -169.5819,B 24.9557,C -1.5391,E1 24.8446,E2 255.8345} C_DIS
LIN {X -119.4404,Y -33.4404,Z 133,A -167.5917,B 24.956,C -1.5317,E1 24.8461,E2 253.8503} C_DIS
LIN {X -118.4229,Y -36.8885,Z 133,A -165.9534,B 24.9564,C -1.5256,E1 24.8474,E2 252.2172} C_DIS
LIN {X -117.2471,Y -40.4654,Z 133,A -164.0338,B 24.9562,C -1.5284,E1 24.8491,E2 250.2799} C_DIS
LIN {X -115.9273,Y -44.1074,Z 133,A -162.4347,B 24.957,C -1.5145,E1 24.8506,E2 248.705} C_DIS
LIN {X -114.938,Y -46.6209,Z 133,A -161.0572,B 24.957,C -1.5167,E1 24.8521,E2 247.3146} C_DIS
LIN {X -112.9855,Y -51.1742,Z 133,A -158.8591,B 24.9575,C -1.5059,E1 24.8545,E2 245.13} C_DIS
LIN {X -111.6547,Y -54.0166,Z 133,A -157.4106,B 24.9578,C -1.5017,E1 24.8563,E2 243.6837} C_DIS
LIN {X -110.1929,Y -56.9422,Z 133,A -155.4283,B 24.9568,C -1.5187,E1 24.8589,E2 241.6502} C_DIS
LIN {X -108.5221,Y -60.0626,Z 133,A -154.1511,B 24.958,C -1.498,E1 24.8605,E2 240.4157} C_DIS
LIN {X -106.4779,Y -63.6172,Z 133,A -152.163,B 24.958,C -1.4971,E1 24.8634,E2 238.4194} C_DIS
LIN {X -104.0433,Y -67.5253,Z 133,A -150.1273,B 24.9586,C -1.4873,E1 24.8664,E2 236.3966} C_DIS
LIN {X -101.995,Y -70.582,Z 133,A -148.3617,B 24.9586,C -1.4859,E1 24.8692,E2 234.6256} C_DIS
LIN {X -99.5933,Y -73.9313,Z 133,A -146.424,B 24.9588,C -1.4827,E1 24.8724,E2 232.6862} C_DIS
LIN {X -97.1423,Y -77.1235,Z 133,A -144.5828,B 24.9591,C -1.4773,E1 24.8755,E2 230.849} C_DIS
LIN {X -95.1088,Y -79.6171,Z 133,A -143.0885,B 24.9593,C -1.4742,E1 24.8782,E2 229.3554} C_DIS
LIN {X -92.4643,Y -82.6742,Z 133,A -141.2223,B 24.9595,C -1.4698,E1 24.8816,E2 227.4912} C_DIS
LIN {X -89.8184,Y -85.5411,Z 133,A -139.3872,B 24.9597,C -1.4673,E1 24.8851,E2 225.6541} C_DIS
LIN {X -86.6754,Y -88.725,Z 133,A -137.3281,B 24.9599,C -1.4625,E1 24.8892,E2 223.5977} C_DIS
LIN {X -83.9889,Y -91.2712,Z 133,A -135.8392,B 24.9607,C -1.4488,E1 24.8922,E2 222.1353} C_DIS
LIN {X -81.8219,Y -93.2193,Z 133,A -134.2902,B 24.9603,C -1.4554,E1 24.8955,E2 220.5644} C_DIS
LIN {X -79.0019,Y -95.6211,Z 133,A -132.5823,B 24.9605,C -1.452,E1 24.8991,E2 218.8581} C_DIS
LIN {X -76.0446,Y -97.9892,Z 133,A -130.6123,B 24.9601,C -1.4589,E1 24.9035,E2 216.8643} C_DIS
LIN {X -73.0539,Y -100.2386,Z 133,A -129.078,B 24.9608,C -1.4469,E1 24.9069,E2 215.3532} C_DIS
LIN {X -69.8763,Y -102.4798,Z 133,A -127.1585,B 24.9606,C -1.4496,E1 24.9113,E2 213.4208} C_DIS
LIN {X -65.9,Y -105.0816,Z 133,A -125.1093,B 24.9612,C -1.4393,E1 24.9161,E2 211.3895} C_DIS
LIN {X -62.9754,Y -106.8585,Z 133,A -123.4309,B 24.9611,C -1.4415,E1 24.9202,E2 209.7006} C_DIS
LIN {X -59.1297,Y -109.0346,Z 133,A -121.3706,B 24.9611,C -1.4396,E1 24.9252,E2 207.6391} C_DIS
LIN {X -55.6937,Y -110.8274,Z 133,A -119.743,B 24.9617,C -1.4297,E1 24.9292,E2 206.0306} C_DIS
LIN {X -53.2727,Y -112.0105,Z 133,A -118.387,B 24.9615,C -1.4334,E1 24.9326,E2 204.6623} C_DIS
LIN {X -49.1048,Y -113.8991,Z 133,A -116.3983,B 24.962,C -1.4251,E1 24.9377,E2 202.6884} C_DIS
LIN {X -46.4796,Y -114.9951,Z 133,A -114.9503,B 24.9617,C -1.4301,E1 24.9414,E2 201.2254} C_DIS
LIN {X -43.3333,Y -116.217,Z 133,A -113.4345,B 24.9619,C -1.4266,E1 24.9454,E2 199.7147} C_DIS
LIN {X -37.2584,Y -118.3065,Z 133,A -110.3895,B 24.9619,C -1.4277,E1 24.9535,E2 196.6613} C_DIS
LIN {X -33.0845,Y -119.5403,Z 133,A -108.362,B 24.9619,C -1.4272,E1 24.9589,E2 194.6318} C_DIS
LIN {X -28.5875,Y -120.6952,Z 133,A -106.3338,B 24.9622,C -1.4204,E1 24.9644,E2 192.6169} C_DIS
LIN {X -25.4958,Y -121.3863,Z 133,A -104.8711,B 24.9622,C -1.4197,E1 24.9684,E2 191.1541} C_DIS
LIN {X -21.6486,Y -122.1295,Z 133,A -103.1397,B 24.9625,C -1.4152,E1 24.9731,E2 189.4314} C_DIS
LIN {X -18.7892,Y -122.6023,Z 133,A -101.6907,B 24.9622,C -1.4201,E1 24.9771,E2 187.9694} C_DIS
LIN {X -15.1656,Y -123.1035,Z 133,A -99.8823,B 24.9619,C -1.4255,E1 24.9822,E2 186.1469} C_DIS
LIN {X -11.3696,Y -123.5126,Z 133,A -98.0548,B 24.9618,C -1.4284,E1 24.9873,E2 184.3115} C_DIS
LIN {X -6.7538,Y -123.8515,Z 133,A -95.9549,B 24.9618,C -1.4266,E1 24.9931,E2 182.2152} C_DIS
LIN {X -2.7431,Y -124.0046,Z 133,A -94.1605,B 24.962,C -1.424,E1 24.9981,E2 180.4268} C_DIS
LIN {X 0.8859,Y -124.0293,Z 133,A -93.2073,B 24.9638,C -1.3894,E1 25.0006,E2 179.5556} C_DIS
Enddeposition()
LIN {X 0.8859,Y -124.0293,Z 133,A -93.2073,B 24.9638,C -1.3894,E1 25.0006,E2 179.5556} C_DIS
Startdeposition()
$VEL.CP = VEL_PRINT
LIN {X -0.0675,Y -123.1989,Z 133,A -93.8487,B 24.9636,C -1.3946,E1 24.9988,E2 180.1847} C_DIS
LIN {X -4.2619,Y -123.1237,Z 133,A -95.792,B 24.9636,C -1.3946,E1 24.9934,E2 182.128} C_DIS
LIN {X -8.2359,Y -122.9224,Z 133,A -97.7799,B 24.9639,C -1.3881,E1 24.9878,E2 184.132} C_DIS
LIN {X -13.016,Y -122.5074,Z 133,A -99.8282,B 24.9634,C -1.397,E1 24.9821,E2 186.1606} C_DIS
LIN {X -16.9419,Y -122.0271,Z 133,A -101.547,B 24.9631,C -1.403,E1 24.9774,E2 187.8663} C_DIS
LIN {X -20.4358,Y -121.4895,Z 133,A -103.6369,B 24.9642,C -1.3826,E1 24.9715,E2 190.0064} C_DIS
LIN {X -23.9849,Y -120.8404,Z 133,A -105.0446,B 24.9635,C -1.3959,E1 24.9677,E2 191.3843} C_DIS
LIN {X -27.768,Y -120.0274,Z 133,A -106.8977,B 24.9635,C -1.3942,E1 24.9627,E2 193.2436} C_DIS
LIN {X -32.936,Y -118.7127,Z 133,A -109.2782,B 24.9633,C -1.4004,E1 24.9563,E2 195.613} C_DIS
LIN {X -36.7255,Y -117.5977,Z 133,A -111.2666,B 24.9636,C -1.3947,E1 24.9509,E2 197.6184} C_DIS
LIN {X -41.3333,Y -116.0571,Z 133,A -113.406,B 24.9632,C -1.4022,E1 24.9453,E2 199.7441} C_DIS
LIN {X -44.5175,Y -114.8721,Z 133,A -114.8926,B 24.9629,C -1.408,E1 24.9415,E2 201.2199} C_DIS
LIN {X -47.9326,Y -113.4899,Z 133,A -117.1212,B 24.964,C -1.3862,E1 24.9356,E2 203.5055} C_DIS
LIN {X -51.5883,Y -111.8745,Z 133,A -118.4018,B 24.9625,C -1.4148,E1 24.9325,E2 204.7212} C_DIS
LIN {X -53.9087,Y -110.7773,Z 133,A -119.9704,B 24.9633,C -1.399,E1 24.9284,E2 206.3314} C_DIS
LIN {X -58.7842,Y -108.2697,Z 133,A -122.3855,B 24.9628,C -1.4086,E1 24.9225,E2 208.7305} C_DIS
LIN {X -62.8547,Y -105.958,Z 133,A -124.55,B 24.9626,C -1.4123,E1 24.9173,E2 210.8926} C_DIS
LIN {X -67.9729,Y -102.7495,Z 133,A -127.3512,B 24.9624,C -1.4171,E1 24.9107,E2 213.6914} C_DIS
LIN {X -70.3817,Y -101.1143,Z 133,A -129.2871,B 24.9636,C -1.3931,E1 24.9062,E2 215.6908} C_DIS
LIN {X -74.3909,Y -98.2027,Z 133,A -131.029,B 24.9621,C -1.4225,E1 24.9024,E2 217.3692} C_DIS
LIN {X -77.046,Y -96.1337,Z 133,A -132.555,B 24.9618,C -1.4272,E1 24.899,E2 218.8897} C_DIS
LIN {X -80.2936,Y -93.4385,Z 133,A -134.5549,B 24.9618,C -1.4293,E1 24.8948,E2 220.8922} C_DIS
LIN {X -83.3607,Y -90.7119,Z 133,A -136.694,B 24.9621,C -1.4229,E1 24.8903,E2 223.0553} C_DIS
LIN {X -85.7027,Y -88.5029,Z 133,A -137.9344,B 24.9613,C -1.4375,E1 24.8879,E2 224.2659} C_DIS
LIN {X -88.4807,Y -85.7257,Z 133,A -139.7507,B 24.961,C -1.442,E1 24.8843,E2 226.0793} C_DIS
LIN {X -91.3836,Y -82.6249,Z 133,A -141.6385,B 24.9606,C -1.4503,E1 24.8808,E2 227.9556} C_DIS
LIN {X -93.6332,Y -80.0675,Z 133,A -143.4428,B 24.9609,C -1.4442,E1 24.8774,E2 229.7828} C_DIS
LIN {X -96.6554,Y -76.3913,Z 133,A -145.6135,B 24.9605,C -1.4514,E1 24.8736,E2 231.9464} C_DIS
LIN {X -98.982,Y -73.3508,Z 133,A -147.4018,B 24.9603,C -1.4555,E1 24.8706,E2 233.7335} C_DIS
LIN {X -101.4047,Y -69.9638,Z 133,A -149.3866,B 24.9602,C -1.4583,E1 24.8674,E2 235.7213} C_DIS
LIN {X -103.1148,Y -67.4195,Z 133,A -151.2295,B 24.961,C -1.4437,E1 24.8646,E2 237.6084} C_DIS
LIN {X -105.3382,Y -63.8871,Z 133,A -152.4058,B 24.9588,C -1.4826,E1 24.863,E2 238.698} C_DIS
LIN {X -109.281,Y -56.8802,Z 133,A -156.5747,B 24.9593,C -1.4738,E1 24.8573,E2 242.9096} C_DIS
LIN {X -111.0088,Y -53.4275,Z 133,A -158.2069,B 24.9586,C -1.4861,E1 24.8553,E2 244.5215} C_DIS
LIN {X -112.0597,Y -51.1873,Z 133,A -160.0047,B 24.96,C -1.4612,E1 24.8531,E2 246.3884} C_DIS
LIN {X -113.9565,Y -46.8154,Z 133,A -162.4507,B 24.9602,C -1.4578,E1 24.8505,E2 248.8562} C_DIS
LIN {X -115.9958,Y -41.503,Z 133,A -164.7093,B 24.9588,C -1.4825,E1 24.8484,E2 251.0687} C_DIS
LIN {X -117.2268,Y -37.8871,Z 133,A -166.0842,B 24.9575,C -1.5054,E1 24.8472,E2 252.3969} C_DIS
LIN {X -118.2899,Y -34.4212,Z 133,A -167.7946,B 24.9573,C -1.5095,E1 24.8459,E2 254.1074} C_DIS
LIN {X -119.3648,Y -30.4857,Z 133,A -169.6705,B 24.9569,C -1.5163,E1 24.8445,E2 255.9779} C_DIS
LIN {X -120.1619,Y -27.1773,Z 133,A -171.3815,B 24.9569,C -1.5157,E1 24.8434,E2 257.7004} C_DIS
LIN {X -121.1422,Y -22.418,Z 133,A -173.6675,B 24.9566,C -1.5217,E1 24.8422,E2 259.9857} C_DIS
LIN {X -121.8709,Y -18.0409,Z 133,A -175.5445,B 24.9558,C -1.5364,E1 24.8414,E2 261.8387} C_DIS
LIN {X -122.5901,Y -12.2222,Z 133,A -179.2038,B 24.9576,C -1.505,E1 24.8403,E2 265.5948} C_DIS
LIN {X -123.0259,Y -6.5057,Z 133,A 179.1058,B 24.9547,C -1.5557,E1 24.84,E2 267.1745} C_DIS
LIN {X -123.1923,Y -1.2278,Z 133,A 176.3454,B 24.955,C -1.5505,E1 24.8398,E2 269.964} C_DIS
LIN {X -122.9836,Y 7.2542,Z 133,A 172.458,B 24.9541,C -1.566,E1 24.8402,E2 273.8378} C_DIS
LIN {X -122.7675,Y 10.2704,Z 133,A 170.8354,B 24.9543,C -1.5613,E1 24.8405,E2 275.4815} C_DIS
LIN {X -121.9895,Y 17.2064,Z 133,A 167.8694,B 24.953,C -1.584,E1 24.8415,E2 278.411} C_DIS
LIN {X -121.4566,Y 20.6326,Z 133,A 166.3751,B 24.9524,C -1.5944,E1 24.8422,E2 279.8894} C_DIS
LIN {X -120.9106,Y 23.6231,Z 133,A 164.5109,B 24.9533,C -1.5795,E1 24.8431,E2 281.8002} C_DIS
LIN {X -119.8594,Y 28.4831,Z 133,A 162.3826,B 24.9523,C -1.5949,E1 24.8444,E2 283.9042} C_DIS
LIN {X -118.9681,Y 32.0019,Z 133,A 160.7071,B 24.952,C -1.6009,E1 24.8456,E2 285.5752} C_DIS
LIN {X -118.0746,Y 35.1562,Z 133,A 158.947,B 24.9523,C -1.5956,E1 24.847,E2 287.3581} C_DIS
LIN {X -116.5435,Y 39.9398,Z 133,A 157.0598,B 24.9507,C -1.6225,E1 24.8486,E2 289.1921} C_DIS
LIN {X -115.5384,Y 42.759,Z 133,A 155.4281,B 24.951,C -1.6164,E1 24.8502,E2 290.8474} C_DIS
LIN {X -114.3724,Y 45.7869,Z 133,A 153.8224,B 24.951,C -1.617,E1 24.8519,E2 292.4608} C_DIS
LIN {X -112.8949,Y 49.3187,Z 133,A 152.0301,B 24.9507,C -1.6219,E1 24.8538,E2 294.2512} C_DIS
LIN {X -111.2716,Y 52.8782,Z 133,A 150.4858,B 24.9496,C -1.6395,E1 24.8556,E2 295.7621} C_DIS
LIN {X -108.5552,Y 58.2542,Z 133,A 147.4843,B 24.9496,C -1.6391,E1 24.8595,E2 298.7806} C_DIS
LIN {X -106.7558,Y 61.4899,Z 133,A 145.6576,B 24.9496,C -1.6396,E1 24.862,E2 300.6156} C_DIS
LIN {X -104.3555,Y 65.4824,Z 133,A 143.5003,B 24.9492,C -1.6463,E1 24.8651,E2 302.7681} C_DIS
LIN {X -100.901,Y 70.6877,Z 133,A 140.5901,B 24.9487,C -1.6543,E1 24.8697,E2 305.6737} C_DIS
LIN {X -98.5323,Y 73.9552,Z 133,A 138.6192,B 24.9487,C -1.6553,E1 24.8729,E2 307.6516} C_DIS
LIN {X -95.6199,Y 77.6831,Z 133,A 136.4728,B 24.9481,C -1.6636,E1 24.8766,E2 309.7884} C_DIS
LIN {X -93.0468,Y 80.747,Z 133,A 134.6014,B 24.9479,C -1.668,E1 24.88,E2 311.6578} C_DIS
LIN {X -90.0818,Y 84.0422,Z 133,A 132.5127,B 24.9476,C -1.6721,E1 24.884,E2 313.7461} C_DIS
LIN {X -87.2368,Y 86.9911,Z 133,A 130.6556,B 24.9472,C -1.6789,E1 24.8876,E2 315.5948} C_DIS
LIN {X -84.1602,Y 89.9722,Z 133,A 128.5543,B 24.9472,C -1.6789,E1 24.8919,E2 317.7048} C_DIS
LIN {X -80.8101,Y 92.9918,Z 133,A 126.5511,B 24.9466,C -1.688,E1 24.896,E2 319.6945} C_DIS
LIN {X -77.7744,Y 95.5454,Z 133,A 124.6522,B 24.9465,C -1.6897,E1 24.9001,E2 321.5964} C_DIS
LIN {X -74.3663,Y 98.2213,Z 133,A 122.6434,B 24.9462,C -1.6943,E1 24.9045,E2 323.6016} C_DIS
LIN {X -71.1711,Y 100.5604,Z 133,A 120.7765,B 24.946,C -1.697,E1 24.9088,E2 325.4685} C_DIS
LIN {X -67.3324,Y 103.1714,Z 133,A 118.8488,B 24.9451,C -1.7116,E1 24.9132,E2 327.368} C_DIS
LIN {X -64.1213,Y 105.196,Z 133,A 116.8816,B 24.9455,C -1.706,E1 24.9179,E2 329.3548} C_DIS
LIN {X -60.6374,Y 107.2428,Z 133,A 114.9382,B 24.9455,C -1.7065,E1 24.9226,E2 331.3027} C_DIS
LIN {X -56.6936,Y 109.3792,Z 133,A 112.9057,B 24.945,C -1.7124,E1 24.9276,E2 333.3267} C_DIS
LIN {X -53.9438,Y 110.7599,Z 133,A 111.1445,B 24.9458,C -1.7,E1 24.9321,E2 335.1221} C_DIS
LIN {X -50.8496,Y 112.2139,Z 133,A 109.8716,B 24.9448,C -1.7166,E1 24.9352,E2 336.3585} C_DIS
LIN {X -47.4508,Y 113.6912,Z 133,A 107.567,B 24.9463,C -1.6931,E1 24.9413,E2 338.7243} C_DIS
LIN {X -43.1404,Y 115.3957,Z 133,A 105.8321,B 24.9449,C -1.7149,E1 24.9457,E2 340.4111} C_DIS
LIN {X -39.0035,Y 116.8588,Z 133,A 103.9723,B 24.9442,C -1.7256,E1 24.9506,E2 342.249} C_DIS
LIN {X -35.302,Y 118.0318,Z 133,A 102.0407,B 24.9444,C -1.722,E1 24.9558,E2 344.1926} C_DIS
LIN {X -31.0519,Y 119.2209,Z 133,A 100.0103,B 24.9442,C -1.7251,E1 24.9612,E2 346.2187} C_DIS
LIN {X -22.4613,Y 121.1343,Z 133,A 95.0148,B 24.9466,C -1.6878,E1 24.9751,E2 351.3086} C_DIS
LIN {X -16.2142,Y 122.125,Z 133,A 93.0603,B 24.9436,C -1.7346,E1 24.9803,E2 353.1536} C_DIS
LIN {X -12.6112,Y 122.5513,Z 133,A 91.2534,B 24.9439,C -1.73,E1 24.9853,E2 354.9725} C_DIS
LIN {X -7.7863,Y 122.9504,Z 133,A 88.8469,B 24.9443,C -1.7239,E1 24.992,E2 357.3945} C_DIS
LIN {X -3.0491,Y 123.1592,Z 133,A 86.8171,B 24.9437,C -1.7327,E1 24.9976,E2 359.4038} C_DIS
LIN {X 0.3886,Y 123.197,Z 133,A 85.0118,B 24.9443,C -1.7234,E1 25.0027,E2 361.2309} C_DIS
LIN {X 4.9833,Y 123.096,Z 133,A 82.8265,B 24.9445,C -1.7214,E1 25.0089,E2 363.4205} C_DIS
LIN {X 8.4002,Y 122.9111,Z 133,A 81.4827,B 24.9437,C -1.7328,E1 25.0125,E2 364.7366} C_DIS
LIN {X 12.286,Y 122.584,Z 133,A 79.6074,B 24.9439,C -1.7297,E1 25.0178,E2 366.6181} C_DIS
LIN {X 16.9358,Y 122.0278,Z 133,A 77.078,B 24.945,C -1.7129,E1 25.0249,E2 369.1854} C_DIS
LIN {X 21.0575,Y 121.3848,Z 133,A 75.5763,B 24.9437,C -1.7327,E1 25.0289,E2 370.6387} C_DIS
LIN {X 24.173,Y 120.8021,Z 133,A 74.0633,B 24.9439,C -1.7302,E1 25.033,E2 372.1556} C_DIS
LIN {X 29.7851,Y 119.5423,Z 133,A 71.4433,B 24.9439,C -1.7313,E1 25.0401,E2 374.7693} C_DIS
LIN {X 33.9907,Y 118.416,Z 133,A 69.3937,B 24.9439,C -1.7287,E1 25.0457,E2 376.8217} C_DIS
LIN {X 38.4396,Y 117.0468,Z 133,A 67.3184,B 24.9439,C -1.7313,E1 25.0512,E2 378.8872} C_DIS
LIN {X 41.5655,Y 115.9732,Z 133,A 65.7366,B 24.9441,C -1.7278,E1 25.0553,E2 380.4742} C_DIS
LIN {X 45.0014,Y 114.6842,Z 133,A 63.6327,B 24.9454,C -1.7072,E1 25.0609,E2 382.6221} C_DIS
LIN {X 48.5655,Y 113.2206,Z 133,A 62.2842,B 24.9441,C -1.7263,E1 25.0643,E2 383.9221} C_DIS
LIN {X 51.739,Y 111.805,Z 133,A 60.4947,B 24.9448,C -1.7162,E1 25.0689,E2 385.7312} C_DIS
LIN {X 55.7646,Y 109.8527,Z 133,A 58.7084,B 24.9441,C -1.7276,E1 25.0733,E2 387.4855} C_DIS
LIN {X 58.8779,Y 108.2184,Z 133,A 56.8864,B 24.9448,C -1.7164,E1 25.0778,E2 389.329} C_DIS
LIN {X 61.694,Y 106.6375,Z 133,A 55.0966,B 24.9458,C -1.7003,E1 25.0822,E2 391.1514} C_DIS
LIN {X 64.7758,Y 104.7947,Z 133,A 53.7309,B 24.945,C -1.7124,E1 25.0854,E2 392.4842} C_DIS
LIN {X 68.0435,Y 102.7029,Z 133,A 52.0576,B 24.9448,C -1.7158,E1 25.0893,E2 394.144} C_DIS
LIN {X 71.8746,Y 100.0596,Z 133,A 49.7368,B 24.9456,C -1.7045,E1 25.0946,E2 396.4834} C_DIS
LIN {X 75.4738,Y 97.3726,Z 133,A 47.7573,B 24.9455,C -1.7061,E1 25.099,E2 398.4521} C_DIS
LIN {X 78.5538,Y 94.9055,Z 133,A 45.8536,B 24.9459,C -1.6992,E1 25.1031,E2 400.3648} C_DIS
LIN {X 81.9645,Y 91.9765,Z 133,A 43.6476,B 24.9465,C -1.6894,E1 25.1078,E2 402.5853} C_DIS
LIN {X 86.7132,Y 87.5131,Z 133,A 40.7697,B 24.9465,C -1.6905,E1 25.1136,E2 405.4488} C_DIS
LIN {X 89.8914,Y 84.247,Z 133,A 38.6597,B 24.9467,C -1.6862,E1 25.1176,E2 407.5598} C_DIS
LIN {X 92.5802,Y 81.2814,Z 133,A 36.9642,B 24.9465,C -1.6901,E1 25.1208,E2 409.2384} C_DIS
LIN {X 94.8655,Y 78.602,Z 133,A 34.9206,B 24.948,C -1.6662,E1 25.1245,E2 411.329} C_DIS
LIN {X 96.9763,Y 75.9828,Z 133,A 33.6122,B 24.9474,C -1.675,E1 25.1267,E2 412.6106} C_DIS
LIN {X 99.4814,Y 72.672,Z 133,A 31.8098,B 24.9474,C -1.6765,E1 25.1297,E2 414.4007} C_DIS
LIN {X 102.2389,Y 68.7384,Z 133,A 29.5385,B 24.9478,C -1.6689,E1 25.1333,E2 416.6789} C_DIS
LIN {X 104.4825,Y 65.2786,Z 133,A 27.5348,B 24.9484,C -1.6595,E1 25.1364,E2 418.6946} C_DIS
LIN {X 106.397,Y 62.1083,Z 133,A 25.8361,B 24.9486,C -1.656,E1 25.1388,E2 420.3928} C_DIS
LIN {X 108.5137,Y 58.3316,Z 133,A 23.8027,B 24.949,C -1.6494,E1 25.1415,E2 422.431} C_DIS
LIN {X 110.4519,Y 54.5675,Z 133,A 22.0294,B 24.9488,C -1.6537,E1 25.1437,E2 424.185} C_DIS
LIN {X 112.672,Y 49.8261,Z 133,A 19.5074,B 24.9495,C -1.6422,E1 25.1467,E2 426.7203} C_DIS
LIN {X 113.9813,Y 46.755,Z 133,A 17.9653,B 24.9497,C -1.6382,E1 25.1483,E2 428.2635} C_DIS
LIN {X 115.6246,Y 42.5287,Z 133,A 15.8283,B 24.9502,C -1.6305,E1 25.1505,E2 430.4068} C_DIS
LIN {X 116.846,Y 39.0421,Z 133,A 14.2335,B 24.9502,C -1.6315,E1 25.1519,E2 431.9902} C_DIS
LIN {X 117.932,Y 35.6316,Z 133,A 12.2628,B 24.9514,C -1.611,E1 25.1536,E2 433.998} C_DIS
LIN {X 118.8358,Y 32.4958,Z 133,A 11.0349,B 24.9508,C -1.6208,E1 25.1544,E2 435.1957} C_DIS
LIN {X 119.6241,Y 29.4556,Z 133,A 8.8599,B 24.9532,C -1.5805,E1 25.156,E2 437.4531} C_DIS
LIN {X 120.772,Y 24.3212,Z 133,A 6.8129,B 24.9525,C -1.5927,E1 25.1571,E2 439.4594} C_DIS
LIN {X 121.4174,Y 20.8668,Z 133,A 5.5486,B 24.9517,C -1.6061,E1 25.1577,E2 440.6849} C_DIS
LIN {X 121.9517,Y 17.4723,Z 133,A 3.9381,B 24.952,C -1.6003,E1 25.1583,E2 442.2995} C_DIS
LIN {X 122.2919,Y 14.9035,Z 133,A 2.5058,B 24.9529,C -1.585,E1 25.1588,E2 443.7594} C_DIS
LIN {X 122.8561,Y 9.1504,Z 133,A 0.1075,B 24.9526,C -1.5909,E1 25.1594,E2 446.1296} C_DIS
LIN {X 123.0771,Y 5.4719,Z 133,A -1.7126,B 24.9532,C -1.5799,E1 25.1597,E2 447.9648} C_DIS
LIN {X 123.1955,Y 0.7179,Z 133,A -3.7731,B 24.9532,C -1.5803,E1 25.1597,E2 450.012} C_DIS
LIN {X 123.1554,Y -3.1842,Z 133,A -5.6503,B 24.9537,C -1.5712,E1 25.1597,E2 451.8996} C_DIS
LIN {X 122.9879,Y -7.1847,Z 133,A -7.528,B 24.9542,C -1.5643,E1 25.1594,E2 453.7824} C_DIS
LIN {X 122.7007,Y -11.0632,Z 133,A -9.1613,B 24.954,C -1.5672,E1 25.1591,E2 455.3991} C_DIS
LIN {X 122.0405,Y -16.8479,Z 133,A -11.9524,B 24.9548,C -1.554,E1 25.1582,E2 458.2046} C_DIS
LIN {X 121.5416,Y -20.1237,Z 133,A -13.3537,B 24.9546,C -1.5561,E1 25.1575,E2 459.5928} C_DIS
LIN {X 120.5772,Y -25.2765,Z 133,A -15.9163,B 24.9555,C -1.5418,E1 25.1562,E2 462.1742} C_DIS
LIN {X 119.2475,Y -30.9465,Z 133,A -18.4982,B 24.9556,C -1.5394,E1 25.1545,E2 464.7467} C_DIS
LIN {X 118.5683,Y -33.4507,Z 133,A -20.5941,B 24.9584,C -1.4908,E1 25.1528,E2 466.9452} C_DIS
LIN {X 116.9221,Y -38.8136,Z 133,A -22.5152,B 24.9569,C -1.517,E1 25.1512,E2 468.7937} C_DIS
LIN {X 115.3855,Y -43.1675,Z 133,A -24.4659,B 24.9567,C -1.5202,E1 25.1494,E2 470.7261} C_DIS
LIN {X 114.1217,Y -46.4073,Z 133,A -26.888,B 24.9593,C -1.4747,E1 25.1467,E2 473.242} C_DIS
LIN {X 111.9622,Y -51.3985,Z 133,A -28.5596,B 24.9573,C -1.5099,E1 25.1449,E2 474.8215} C_DIS
LIN {X 110.5516,Y -54.3656,Z 133,A -30.1369,B 24.9577,C -1.5027,E1 25.143,E2 476.4073} C_DIS
LIN {X 108.3514,Y -58.6342,Z 133,A -32.7401,B 24.9591,C -1.4774,E1 25.1395,E2 479.0565} C_DIS
LIN {X 106.6626,Y -61.6507,Z 133,A -34.0375,B 24.9585,C -1.4882,E1 25.1378,E2 480.3216} C_DIS
LIN {X 104.3909,Y -65.426,Z 133,A -36.1412,B 24.959,C -1.4795,E1 25.1347,E2 482.4352} C_DIS
LIN {X 101.7507,Y -69.4598,Z 133,A -38.3158,B 24.9592,C -1.4765,E1 25.1313,E2 484.6061} C_DIS
LIN {X 99.4029,Y -72.7789,Z 133,A -40.0359,B 24.959,C -1.4798,E1 25.1286,E2 486.31} C_DIS
LIN {X 95.2753,Y -78.1045,Z 133,A -43.3576,B 24.96,C -1.4618,E1 25.1228,E2 489.6585} C_DIS
LIN {X 93.3589,Y -80.3859,Z 133,A -45.3368,B 24.9618,C -1.4286,E1 25.1191,E2 491.7071} C_DIS
LIN {X 89.8115,Y -84.3319,Z 133,A -46.8939,B 24.9597,C -1.4676,E1 25.1163,E2 493.1655} C_DIS
LIN {X 85.4971,Y -88.7016,Z 133,A -49.9037,B 24.9605,C -1.4527,E1 25.1103,E2 496.1975} C_DIS
LIN {X 80.5311,Y -93.2336,Z 133,A -53.5401,B 24.9622,C -1.4201,E1 25.1026,E2 499.8964} C_DIS
LIN {X 77.2555,Y -95.9649,Z 133,A -54.9024,B 24.9608,C -1.4464,E1 25.0998,E2 501.1915} C_DIS
LIN {X 71.7819,Y -100.1258,Z 133,A -58.6239,B 24.9626,C -1.4136,E1 25.0913,E2 504.9771} C_DIS
LIN {X 68.5738,Y -102.349,Z 133,A -59.9893,B 24.9616,C -1.4321,E1 25.0883,E2 506.2942} C_DIS
LIN {X 65.2813,Y -104.4807,Z 133,A -61.5681,B 24.9611,C -1.4406,E1 25.0846,E2 507.8477} C_DIS
LIN {X 61.9577,Y -106.484,Z 133,A -63.6264,B 24.962,C -1.4247,E1 25.0796,E2 509.9373} C_DIS
LIN {X 58.1929,Y -108.588,Z 133,A -65.6755,B 24.9623,C -1.419,E1 25.0745,E2 511.9939} C_DIS
LIN {X 54.5884,Y -110.4416,Z 133,A -67.9645,B 24.9635,C -1.3961,E1 25.0687,E2 514.3307} C_DIS
LIN {X 50.7835,Y -112.2435,Z 133,A -69.4337,B 24.9624,C -1.4169,E1 25.0651,E2 515.7472} C_DIS
LIN {X 47.603,Y -113.6276,Z 133,A -71.0447,B 24.9625,C -1.4146,E1 25.061,E2 517.3598} C_DIS
LIN {X 43.8688,Y -115.123,Z 133,A -72.832,B 24.9625,C -1.416,E1 25.0563,E2 519.1398} C_DIS
LIN {X 39.6166,Y -116.6545,Z 133,A -75.1,B 24.963,C -1.4051,E1 25.0503,E2 521.4289} C_DIS
LIN {X 35.9582,Y -117.8322,Z 133,A -76.7788,B 24.9628,C -1.4083,E1 25.0459,E2 523.0972} C_DIS
LIN {X 28.4476,Y -119.868,Z 133,A -80.4959,B 24.9633,C -1.3997,E1 25.0358,E2 526.8289} C_DIS
LIN {X 24.5142,Y -120.7327,Z 133,A -82.9283,B 24.9648,C -1.3712,E1 25.029,E2 529.3257} C_DIS
LIN {X 19.5166,Y -121.6425,Z 133,A -84.7245,B 24.9635,C -1.3964,E1 25.0242,E2 531.0604} C_DIS
LIN {X 13.9156,Y -122.4096,Z 133,A -87.3012,B 24.9635,C -1.3972,E1 25.0171,E2 533.6331} C_DIS
LIN {X 10.2213,Y -122.7717,Z 133,A -88.9707,B 24.9633,C -1.3991,E1 25.0124,E2 535.2973} C_DIS
LIN {X 7.1244,Y -122.9916,Z 133,A -90.6361,B 24.9639,C -1.3878,E1 25.0077,E2 536.9885} C_DIS
LIN {X 1.8852,Y -123.1822,Z 133,A -92.8232,B 24.9633,C -1.399,E1 25.0017,E2 539.1487} C_DIS
LIN {X 1.8852,Y -123.1822,Z 133,A -92.8232,B 24.9633,C -1.399,E1 25.0017,E2 539.1487} C_DIS
Enddeposition()
LIN {X 0.8729,Y -122.3542,Z 133,A -92.9863,B 24.9618,C -1.4283,E1 25.0014,E2 539.2424} C_DIS
Startdeposition()
$VEL.CP = VEL_PRINT
LIN {X 5.1349,Y -122.2527,Z 133,A -90.4329,B 24.9603,C -1.4556,E1 25.0087,E2 536.625} C_DIS
LIN {X 10.0121,Y -121.9494,Z 133,A -88.3393,B 24.9608,C -1.4473,E1 25.0145,E2 534.552} C_DIS
LIN {X 13.5028,Y -121.6129,Z 133,A -85.9618,B 24.9587,C -1.4839,E1 25.0214,E2 532.0893} C_DIS
LIN {X 18.6304,Y -120.9332,Z 133,A -84.5812,B 24.9614,C -1.435,E1 25.0248,E2 530.8258} C_DIS
LIN {X 24.8228,Y -119.8159,Z 133,A -81.2899,B 24.9604,C -1.454,E1 25.034,E2 527.4931} C_DIS
LIN {X 32.1123,Y -118.0721,Z 133,A -77.6574,B 24.9599,C -1.4635,E1 25.0439,E2 523.8436} C_DIS
LIN {X 35.7568,Y -117.0187,Z 133,A -76.0344,B 24.9602,C -1.4581,E1 25.0482,E2 522.2363} C_DIS
LIN {X 39.1256,Y -115.9361,Z 133,A -74.4683,B 24.9603,C -1.4557,E1 25.0523,E2 520.6788} C_DIS
LIN {X 44.7917,Y -113.8678,Z 133,A -71.6608,B 24.9601,C -1.4587,E1 25.0597,E2 517.8702} C_DIS
LIN {X 47.3846,Y -112.8119,Z 133,A -70.3328,B 24.96,C -1.4615,E1 25.0631,E2 516.5387} C_DIS
LIN {X 54.7382,Y -109.4343,Z 133,A -66.5924,B 24.9598,C -1.465,E1 25.0726,E2 512.7995} C_DIS
LIN {X 56.9677,Y -108.2892,Z 133,A -65.3158,B 24.9594,C -1.4721,E1 25.0757,E2 511.5097} C_DIS
LIN {X 63.3684,Y -104.674,Z 133,A -61.9789,B 24.9594,C -1.4731,E1 25.0838,E2 508.1803} C_DIS
LIN {X 66.0015,Y -103.0338,Z 133,A -60.4271,B 24.9589,C -1.4809,E1 25.0875,E2 506.6153} C_DIS
LIN {X 69.1611,Y -100.9407,Z 133,A -58.4085,B 24.958,C -1.4967,E1 25.0922,E2 504.5662} C_DIS
LIN {X 74.9737,Y -96.7015,Z 133,A -55.5127,B 24.959,C -1.4802,E1 25.0986,E2 501.7196} C_DIS
LIN {X 77.3559,Y -94.8068,Z 133,A -53.3303,B 24.9566,C -1.5214,E1 25.1035,E2 499.4482} C_DIS
LIN {X 80.8008,Y -91.8882,Z 133,A -51.1468,B 24.9561,C -1.5299,E1 25.1081,E2 497.2534} C_DIS
LIN {X 84.4179,Y -88.5766,Z 133,A -49.5251,B 24.9578,C -1.5014,E1 25.1113,E2 495.7056} C_DIS
LIN {X 89.5231,Y -83.414,Z 133,A -45.6085,B 24.9558,C -1.536,E1 25.119,E2 491.7242} C_DIS
LIN {X 92.389,Y -80.2281,Z 133,A -44.3585,B 24.9577,C -1.503,E1 25.1212,E2 490.5577} C_DIS
LIN {X 94.4429,Y -77.8009,Z 133,A -41.9028,B 24.9546,C -1.556,E1 25.1257,E2 487.9884} C_DIS
LIN {X 97.7702,Y -73.5755,Z 133,A -40.3254,B 24.957,C -1.5151,E1 25.1282,E2 486.5149} C_DIS
LIN {X 99.5656,Y -71.1263,Z 133,A -38.6534,B 24.956,C -1.5317,E1 25.131,E2 484.8119} C_DIS
LIN {X 102.0044,Y -67.5827,Z 133,A -36.6695,B 24.9558,C -1.5358,E1 25.1341,E2 482.828} C_DIS
LIN {X 104.1195,Y -64.2766,Z 133,A -34.8444,B 24.9555,C -1.5405,E1 25.1368,E2 481.0011} C_DIS
LIN {X 106.3078,Y -60.5883,Z 133,A -32.3793,B 24.9538,C -1.5698,E1 25.1403,E2 478.4798} C_DIS
LIN {X 108.3481,Y -56.8558,Z 133,A -30.3951,B 24.9535,C -1.5754,E1 25.1429,E2 476.4927} C_DIS
LIN {X 110.3097,Y -52.9497,Z 133,A -29.2064,B 24.9557,C -1.5379,E1 25.1443,E2 475.3987} C_DIS
LIN {X 112.7059,Y -47.6382,Z 133,A -26.1129,B 24.9541,C -1.5648,E1 25.1478,E2 472.2587} C_DIS
LIN {X 114.0407,Y -44.3466,Z 133,A -24.5614,B 24.9541,C -1.5643,E1 25.1494,E2 470.7169} C_DIS
LIN {X 115.2735,Y -41.0392,Z 133,A -22.9652,B 24.9541,C -1.5667,E1 25.1509,E2 469.1242} C_DIS
LIN {X 117.6664,Y -33.5677,Z 133,A -19.3944,B 24.9536,C -1.5731,E1 25.1539,E2 465.5585} C_DIS
LIN {X 118.4452,Y -30.7076,Z 133,A -17.0991,B 24.9506,C -1.624,E1 25.1556,E2 463.1564} C_DIS
LIN {X 119.6889,Y -25.4273,Z 133,A -14.5406,B 24.95,C -1.6332,E1 25.157,E2 460.5911} C_DIS
LIN {X 120.7294,Y -19.9068,Z 133,A -12.7441,B 24.9521,C -1.599,E1 25.1579,E2 458.8857} C_DIS
LIN {X 121.8793,Y -10.8466,Z 133,A -8.4385,B 24.9512,C -1.6144,E1 25.1593,E2 454.5694} C_DIS
LIN {X 122.1416,Y -7.3105,Z 133,A -6.8776,B 24.9512,C -1.6148,E1 25.1596,E2 453.0167} C_DIS
LIN {X 122.2988,Y -3.8807,Z 133,A -4.9332,B 24.9498,C -1.6373,E1 25.1598,E2 451.0309} C_DIS
LIN {X 122.3592,Y -0.6047,Z 133,A -3.8436,B 24.9508,C -1.6196,E1 25.1598,E2 449.9894} C_DIS
LIN {X 122.2721,Y 4.6285,Z 133,A -1.3259,B 24.9502,C -1.631,E1 25.1596,E2 447.4598} C_DIS
LIN {X 122.0835,Y 8.2413,Z 133,A 0.8759,B 24.9482,C -1.6624,E1 25.1592,E2 445.1971} C_DIS
LIN {X 121.7419,Y 12.2986,Z 133,A 2.8984,B 24.9475,C -1.6746,E1 25.1586,E2 443.158} C_DIS
LIN {X 121.1895,Y 16.8881,Z 133,A 4.2141,B 24.9497,C -1.6383,E1 25.1582,E2 441.9356} C_DIS
LIN {X 120.7629,Y 19.7065,Z 133,A 6.51,B 24.9464,C -1.6915,E1 25.1571,E2 439.5276} C_DIS
LIN {X 119.7858,Y 24.9704,Z 133,A 9.0007,B 24.9459,C -1.6986,E1 25.1557,E2 437.0346} C_DIS
LIN {X 118.6016,Y 30.0907,Z 133,A 10.3213,B 24.9491,C -1.6484,E1 25.1549,E2 435.8402} C_DIS
LIN {X 117.0899,Y 35.5237,Z 133,A 13.0612,B 24.9483,C -1.6615,E1 25.1528,E2 433.085} C_DIS
LIN {X 116.2158,Y 38.2861,Z 133,A 14.7224,B 24.947,C -1.681,E1 25.1514,E2 431.3873} C_DIS
LIN {X 115.0123,Y 41.7627,Z 133,A 16.3865,B 24.947,C -1.6832,E1 25.1498,E2 429.7273} C_DIS
LIN {X 113.4249,Y 45.8981,Z 133,A 18.4476,B 24.9466,C -1.6888,E1 25.1477,E2 427.6645} C_DIS
LIN {X 112.0331,Y 49.2031,Z 133,A 20.3033,B 24.9457,C -1.7025,E1 25.1456,E2 425.7866} C_DIS
LIN {X 109.7658,Y 54.0669,Z 133,A 22.6263,B 24.9458,C -1.7002,E1 25.1429,E2 423.4815} C_DIS
LIN {X 108.1133,Y 57.3019,Z 133,A 24.2915,B 24.9456,C -1.7032,E1 25.1407,E2 421.8181} C_DIS
LIN {X 106.1554,Y 60.855,Z 133,A 26.3804,B 24.9447,C -1.7179,E1 25.1378,E2 419.7053} C_DIS
LIN {X 104.3414,Y 63.9144,Z 133,A 27.8818,B 24.9449,C -1.7142,E1 25.1357,E2 418.2204} C_DIS
LIN {X 102.2217,Y 67.2534,Z 133,A 30.2315,B 24.943,C -1.744,E1 25.132,E2 415.812} C_DIS
LIN {X 99.7562,Y 70.8595,Z 133,A 31.4789,B 24.9452,C -1.7093,E1 25.1301,E2 414.6526} C_DIS
LIN {X 97.259,Y 74.2489,Z 133,A 33.72,B 24.9441,C -1.7277,E1 25.1263,E2 412.3789} C_DIS
LIN {X 93.4742,Y 78.9612,Z 133,A 36.2305,B 24.9446,C -1.7186,E1 25.122,E2 409.9015} C_DIS
LIN {X 91.5514,Y 81.1825,Z 133,A 37.9126,B 24.9435,C -1.737,E1 25.1188,E2 408.1835} C_DIS
LIN {X 88.8387,Y 84.1424,Z 133,A 39.7866,B 24.9432,C -1.7409,E1 25.1152,E2 406.3085} C_DIS
LIN {X 85.8762,Y 87.1642,Z 133,A 42.3516,B 24.941,C -1.7742,E1 25.11,E2 403.6756} C_DIS
LIN {X 82.3979,Y 90.4589,Z 133,A 43.6175,B 24.9439,C -1.7305,E1 25.1077,E2 402.5181} C_DIS
LIN {X 80.2914,Y 92.3337,Z 133,A 45.3049,B 24.9425,C -1.7512,E1 25.104,E2 400.7886} C_DIS
LIN {X 77.2151,Y 94.9217,Z 133,A 47.2043,B 24.9422,C -1.7557,E1 25.0999,E2 398.8859} C_DIS
LIN {X 73.5973,Y 97.7536,Z 133,A 49.3758,B 24.9419,C -1.7606,E1 25.0951,E2 396.7107} C_DIS
LIN {X 70.4752,Y 100.0271,Z 133,A 51.6703,B 24.9401,C -1.7876,E1 25.0898,E2 394.3603} C_DIS
LIN {X 66.6636,Y 102.6074,Z 133,A 53.2414,B 24.9418,C -1.7625,E1 25.0863,E2 392.8539} C_DIS
LIN {X 60.7253,Y 106.2295,Z 133,A 56.1215,B 24.9427,C -1.7491,E1 25.0795,E2 390.0143} C_DIS
LIN {X 56.3192,Y 108.6305,Z 133,A 58.7995,B 24.9414,C -1.7682,E1 25.0728,E2 387.2988} C_DIS
LIN {X 53.5439,Y 110.0241,Z 133,A 60.778,B 24.9396,C -1.7955,E1 25.0677,E2 385.2611} C_DIS
LIN {X 49.8404,Y 111.7487,Z 133,A 61.9543,B 24.9418,C -1.7621,E1 25.0649,E2 384.1667} C_DIS
LIN {X 43.7518,Y 114.2718,Z 133,A 65.2085,B 24.9411,C -1.7733,E1 25.0564,E2 380.8934} C_DIS
LIN {X 41.1588,Y 115.2303,Z 133,A 66.5973,B 24.9407,C -1.779,E1 25.0528,E2 379.4939} C_DIS
LIN {X 37.4931,Y 116.4742,Z 133,A 68.6511,B 24.9398,C -1.7921,E1 25.0472,E2 377.4131} C_DIS
LIN {X 33.3897,Y 117.7163,Z 133,A 70.3491,B 24.9407,C -1.7787,E1 25.0428,E2 375.7496} C_DIS
LIN {X 30.1192,Y 118.5943,Z 133,A 71.9586,B 24.9406,C -1.7809,E1 25.0384,E2 374.1374} C_DIS
LIN {X 25.281,Y 119.72,Z 133,A 74.7909,B 24.9388,C -1.8062,E1 25.0305,E2 371.2489} C_DIS
LIN {X 21.1259,Y 120.5226,Z 133,A 76.1424,B 24.9408,C -1.777,E1 25.027,E2 369.9681} C_DIS
LIN {X 17.387,Y 121.1186,Z 133,A 78.1657,B 24.94,C -1.7894,E1 25.0214,E2 367.9174} C_DIS
LIN {X 11.1424,Y 121.853,Z 133,A 81.0955,B 24.94,C -1.7891,E1 25.0132,E2 364.9902} C_DIS
LIN {X 3.9446,Y 122.297,Z 133,A 84.1911,B 24.9409,C -1.7758,E1 25.0047,E2 361.9273} C_DIS
LIN {X -1.2238,Y 122.3554,Z 133,A 86.7034,B 24.9406,C -1.7796,E1 24.9977,E2 359.406} C_DIS
LIN {X -4.555,Y 122.275,Z 133,A 88.8866,B 24.9387,C -1.8083,E1 24.9914,E2 357.1544} C_DIS
LIN {X -8.9505,Y 122.0316,Z 133,A 90.2964,B 24.9408,C -1.777,E1 24.9877,E2 355.8183} C_DIS
LIN {X -14.8238,Y 121.4586,Z 133,A 93.088,B 24.9408,C -1.7768,E1 24.9799,E2 353.0256} C_DIS
LIN {X -22.8289,Y 120.2118,Z 133,A 96.6877,B 24.9416,C -1.7651,E1 24.9701,E2 349.4505} C_DIS
LIN {X -28.0283,Y 119.1084,Z 133,A 99.3887,B 24.9411,C -1.7725,E1 24.9626,E2 346.7284} C_DIS
LIN {X -32.1636,Y 118.059,Z 133,A 101.6169,B 24.9405,C -1.7811,E1 24.9565,E2 344.4768} C_DIS
LIN {X -35.9989,Y 116.9447,Z 133,A 103.3236,B 24.9412,C -1.7715,E1 24.952,E2 342.7899} C_DIS
LIN {X -39.1107,Y 115.941,Z 133,A 104.9246,B 24.9411,C -1.7728,E1 24.9477,E2 341.1827} C_DIS
LIN {X -47.4108,Y 112.801,Z 133,A 108.9923,B 24.9417,C -1.7631,E1 24.9372,E2 337.1295} C_DIS
LIN {X -50.9806,Y 111.2334,Z 133,A 110.8595,B 24.9418,C -1.7622,E1 24.9324,E2 335.26} C_DIS
LIN {X -54.3928,Y 109.6049,Z 133,A 112.6281,B 24.942,C -1.7593,E1 24.928,E2 333.4937} C_DIS
LIN {X -57.6793,Y 107.9137,Z 133,A 114.409,B 24.942,C -1.7586,E1 24.9236,E2 331.7096} C_DIS
LIN {X -60.9599,Y 106.0955,Z 133,A 116.2236,B 24.942,C -1.758,E1 24.9192,E2 329.8909} C_DIS
LIN {X -66.9902,Y 102.3954,Z 133,A 119.5697,B 24.9424,C -1.7532,E1 24.9113,E2 326.5458} C_DIS
LIN {X -70.475,Y 100.0272,Z 133,A 121.4941,B 24.9428,C -1.747,E1 24.9068,E2 324.6295} C_DIS
LIN {X -73.7859,Y 97.611,Z 133,A 123.4674,B 24.9429,C -1.7454,E1 24.9024,E2 322.6531} C_DIS
LIN {X -77.2441,Y 94.898,Z 133,A 125.519,B 24.9432,C -1.7406,E1 24.898,E2 320.6053} C_DIS
LIN {X -80.317,Y 92.3113,Z 133,A 127.3776,B 24.9436,C -1.7353,E1 24.894,E2 318.752} C_DIS
LIN {X -83.5633,Y 89.3844,Z 133,A 129.4998,B 24.9436,C -1.7338,E1 24.8896,E2 316.6248} C_DIS
LIN {X -86.635,Y 86.4094,Z 133,A 131.4672,B 24.9441,C -1.7274,E1 24.8858,E2 314.6644} C_DIS
LIN {X -89.5808,Y 83.352,Z 133,A 133.4875,B 24.9443,C -1.7238,E1 24.8819,E2 312.6438} C_DIS
LIN {X -92.4987,Y 80.1018,Z 133,A 135.5421,B 24.9446,C -1.7189,E1 24.8781,E2 310.5915} C_DIS
LIN {X -95.0818,Y 77.0176,Z 133,A 137.4157,B 24.945,C -1.7135,E1 24.8748,E2 308.7223} C_DIS
LIN {X -97.8334,Y 73.4919,Z 133,A 139.5944,B 24.9451,C -1.7115,E1 24.8711,E2 306.5379} C_DIS
LIN {X -100.6587,Y 69.5719,Z 133,A 142.6492,B 24.9432,C -1.7404,E1 24.8661,E2 303.3993} C_DIS
LIN {X -103.9716,Y 64.515,Z 133,A 144.4054,B 24.9468,C -1.6846,E1 24.8636,E2 301.7669} C_DIS
LIN {X -105.3943,Y 62.1636,Z 133,A 145.9623,B 24.9463,C -1.6927,E1 24.8614,E2 300.1827} C_DIS
LIN {X -109.9956,Y 53.6016,Z 133,A 150.3933,B 24.9475,C -1.6737,E1 24.8556,E2 295.7735} C_DIS
LIN {X -111.5402,Y 50.3064,Z 133,A 152.2035,B 24.9475,C -1.6732,E1 24.8535,E2 293.9547} C_DIS
LIN {X -112.8892,Y 47.1996,Z 133,A 153.7386,B 24.948,C -1.6661,E1 24.8518,E2 292.4281} C_DIS
LIN {X -114.0346,Y 44.3624,Z 133,A 155.2241,B 24.9481,C -1.6639,E1 24.8503,E2 290.9394} C_DIS
LIN {X -115.2262,Y 41.1704,Z 133,A 156.8989,B 24.9482,C -1.6623,E1 24.8487,E2 289.2589} C_DIS
LIN {X -117.1942,Y 35.1827,Z 133,A 159.8444,B 24.9488,C -1.6526,E1 24.8462,E2 286.3195} C_DIS
LIN {X -118.1672,Y 31.7574,Z 133,A 161.4847,B 24.9492,C -1.6461,E1 24.845,E2 284.6852} C_DIS
LIN {X -119.0312,Y 28.3476,Z 133,A 163.2152,B 24.9493,C -1.6445,E1 24.8438,E2 282.9486} C_DIS
LIN {X -120.2682,Y 22.5351,Z 133,A 165.9646,B 24.95,C -1.6339,E1 24.8423,E2 280.2081} C_DIS
LIN {X -120.897,Y 18.8639,Z 133,A 167.6601,B 24.9505,C -1.6261,E1 24.8415,E2 278.5211} C_DIS
LIN {X -121.3817,Y 15.4453,Z 133,A 169.5348,B 24.9501,C -1.6321,E1 24.8408,E2 276.6209} C_DIS
LIN {X -122.0935,Y 8.0825,Z 133,A 172.6415,B 24.9517,C -1.6051,E1 24.8401,E2 273.56} C_DIS
LIN {X -122.355,Y 1.2935,Z 133,A 175.8773,B 24.9522,C -1.597,E1 24.8398,E2 270.3241} C_DIS
LIN {X -122.2802,Y -4.4199,Z 133,A 178.4542,B 24.953,C -1.5839,E1 24.8399,E2 267.7628} C_DIS
LIN {X -122.0851,Y -8.2169,Z 133,A -178.9426,B 24.9512,C -1.6141,E1 24.8404,E2 265.0718} C_DIS
LIN {X -121.7118,Y -12.59,Z 133,A -177.0239,B 24.9519,C -1.6015,E1 24.8409,E2 263.1719} C_DIS
LIN {X -121.2891,Y -16.1523,Z 133,A -175.8074,B 24.9535,C -1.5757,E1 24.8413,E2 262.0095} C_DIS
LIN {X -120.7958,Y -19.5091,Z 133,A -173.9356,B 24.953,C -1.583,E1 24.8422,E2 260.1091} C_DIS
LIN {X -120.1373,Y -23.217,Z 133,A -172.3714,B 24.9539,C -1.5687,E1 24.8429,E2 258.5698} C_DIS
LIN {X -119.3208,Y -27.1016,Z 133,A -170.526,B 24.9543,C -1.5623,E1 24.844,E2 256.7289} C_DIS
LIN {X -118.557,Y -30.2664,Z 133,A -168.9595,B 24.9544,C -1.5593,E1 24.8451,E2 255.1602} C_DIS
LIN {X -117.4269,Y -34.3905,Z 133,A -166.9628,B 24.9548,C -1.5529,E1 24.8466,E2 253.1672} C_DIS
LIN {X -116.4255,Y -37.6454,Z 133,A -164.7467,B 24.9535,C -1.5755,E1 24.8486,E2 250.8846} C_DIS
LIN {X -114.9434,Y -41.9538,Z 133,A -162.9736,B 24.9548,C -1.5531,E1 24.8502,E2 249.1548} C_DIS
LIN {X -113.4305,Y -45.8843,Z 133,A -161.1793,B 24.9556,C -1.5394,E1 24.852,E2 247.3832} C_DIS
LIN {X -111.1539,Y -51.1527,Z 133,A -158.5475,B 24.9562,C -1.5291,E1 24.855,E2 244.7614} C_DIS
LIN {X -109.7436,Y -54.1118,Z 133,A -156.9535,B 24.9562,C -1.5273,E1 24.8569,E2 243.163} C_DIS
LIN {X -108.3283,Y -56.8934,Z 133,A -154.5592,B 24.9541,C -1.565,E1 24.8602,E2 240.6663} C_DIS
LIN {X -105.2974,Y -62.3286,Z 133,A -152.4558,B 24.9567,C -1.5206,E1 24.863,E2 238.6577} C_DIS
LIN {X -102.2233,Y -67.2509,Z 133,A -149.8985,B 24.9575,C -1.5063,E1 24.8668,E2 236.1216} C_DIS
LIN {X -100.5232,Y -69.7664,Z 133,A -148.3171,B 24.9573,C -1.5097,E1 24.8693,E2 234.5241} C_DIS
LIN {X -97.7783,Y -73.5648,Z 133,A -146.1256,B 24.9576,C -1.5041,E1 24.873,E2 232.3355} C_DIS
LIN {X -94.5407,Y -77.6821,Z 133,A -143.6621,B 24.9579,C -1.4986,E1 24.8773,E2 229.8734} C_DIS
LIN {X -92.0474,Y -80.6193,Z 133,A -141.7729,B 24.9579,C -1.4983,E1 24.8807,E2 227.9765} C_DIS
LIN {X -89.2126,Y -83.7473,Z 133,A -139.8127,B 24.9582,C -1.4931,E1 24.8844,E2 226.02} C_DIS
LIN {X -86.152,Y -86.8909,Z 133,A -137.2282,B 24.9571,C -1.5128,E1 24.8897,E2 223.3777} C_DIS
LIN {X -82.7324,Y -90.1527,Z 133,A -135.9148,B 24.9597,C -1.4673,E1 24.8921,E2 222.1671} C_DIS
LIN {X -79.4237,Y -93.0819,Z 133,A -133.565,B 24.9592,C -1.4759,E1 24.8971,E2 219.7878} C_DIS
LIN {X -76.3153,Y -95.646,Z 133,A -131.8526,B 24.9598,C -1.4644,E1 24.9008,E2 218.0961} C_DIS
LIN {X -73.9225,Y -97.5076,Z 133,A -130.171,B 24.9593,C -1.4737,E1 24.9046,E2 216.3863} C_DIS
LIN {X -68.2201,Y -101.579,Z 133,A -127.1306,B 24.9602,C -1.4571,E1 24.9114,E2 213.3749} C_DIS
LIN {X -64.1041,Y -104.2252,Z 133,A -124.8903,B 24.9606,C -1.4511,E1 24.9167,E2 211.1416} C_DIS
LIN {X -61.6911,Y -105.6715,Z 133,A -123.2359,B 24.9598,C -1.4647,E1 24.9208,E2 209.4501} C_DIS
LIN {X -57.9536,Y -107.7669,Z 133,A -121.1663,B 24.9598,C -1.4648,E1 24.9258,E2 207.3742} C_DIS
LIN {X -52.0787,Y -110.726,Z 133,A -117.3474,B 24.9581,C -1.4956,E1 24.9357,E2 203.4724} C_DIS
LIN {X -46.7499,Y -113.077,Z 133,A -116.0035,B 24.9618,C -1.4282,E1 24.9387,E2 202.2855} C_DIS
LIN {X -42.9796,Y -114.5623,Z 133,A -113.5611,B 24.9605,C -1.4515,E1 24.9452,E2 199.7823} C_DIS
LIN {X -37.8207,Y -116.3694,Z 133,A -110.9764,B 24.9605,C -1.4505,E1 24.9521,E2 197.1952} C_DIS
LIN {X -34.2537,Y -117.4669,Z 133,A -109.3281,B 24.9609,C -1.4446,E1 24.9564,E2 195.558} C_DIS
LIN {X -30.821,Y -118.4162,Z 133,A -107.4332,B 24.9604,C -1.4542,E1 24.9616,E2 193.6375} C_DIS
LIN {X -24.1915,Y -119.9444,Z 133,A -103.7277,B 24.9591,C -1.4775,E1 24.9719,E2 189.8724} C_DIS
LIN {X -19.2112,Y -120.8431,Z 133,A -102.1058,B 24.9611,C -1.4411,E1 24.9761,E2 188.3351} C_DIS
LIN {X -15.299,Y -121.4008,Z 133,A -100.0918,B 24.9607,C -1.4485,E1 24.9818,E2 186.3022} C_DIS
LIN {X -11.5235,Y -121.8165,Z 133,A -97.9147,B 24.9597,C -1.4674,E1 24.9879,E2 184.0791} C_DIS
LIN {X -7.4469,Y -122.1331,Z 133,A -96.619,B 24.9613,C -1.4378,E1 24.9914,E2 182.8529} C_DIS
LIN {X -2.9516,Y -122.3248,Z 133,A -94.4966,B 24.9613,C -1.4388,E1 24.9973,E2 180.728} C_DIS
LIN {X -0.1714,Y -122.3614,Z 133,A -93.0303,B 24.9608,C -1.4469,E1 25.0014,E2 179.2424} C_DIS
Enddeposition()
END
